Yaskawa INFORM job: A_ROOF_SIDE_0617_2_PAINT_55.JBI

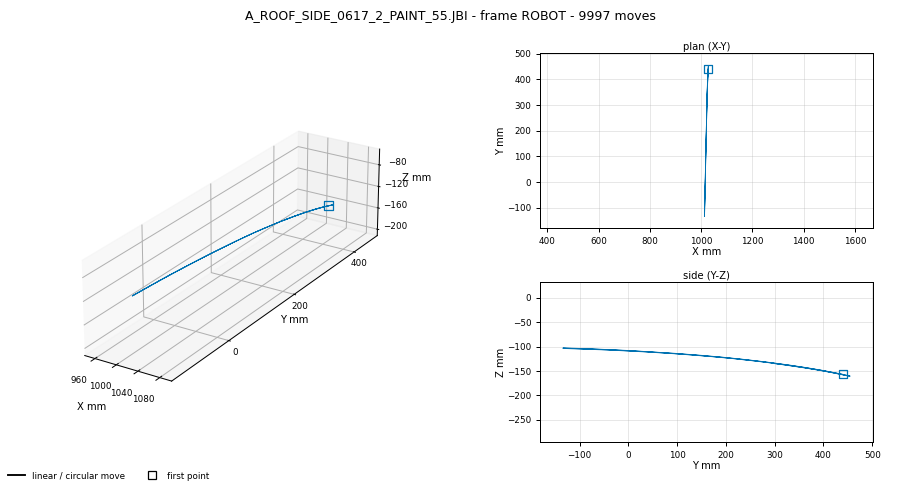
[picture p0: tool path of A_ROOF_SIDE_0617_2_PAINT_55.JBI in frame ROBOT, 9997 of 9997 moves have a stored position in this frame; points joined in program order, loops and branches not executed]
/JOB
//NAME A_ROOF_SIDE_0617_2_PAINT55
//POS
///NPOS 9997,0,0,0,0,0
///TOOL 1
///USER 0
///POSTYPE ROBOT
///RECTAN
///RCONF 1,0,0,0,0,0,0,0,0,0,0,0,0,0,0,0,0,0,0,0,0,0,0,0
C00000=1028.136,439.108,-156.615,175.575,49.117,160.317
C00001=1028.123,438.864,-156.563,175.557,49.112,160.312
C00002=1028.110,438.620,-156.510,175.540,49.107,160.308
C00003=1028.096,438.376,-156.458,175.523,49.102,160.304
C00004=1028.083,438.132,-156.405,175.506,49.097,160.300
C00005=1028.070,437.888,-156.353,175.488,49.092,160.296
C00006=1028.056,437.643,-156.301,175.472,49.087,160.291
C00007=1028.043,437.399,-156.249,175.455,49.082,160.287
C00008=1028.030,437.155,-156.196,175.437,49.078,160.283
C00009=1028.016,436.911,-156.144,175.421,49.072,160.279
C00010=1028.003,436.666,-156.092,175.404,49.067,160.275
C00011=1027.990,436.423,-156.040,175.387,49.063,160.271
C00012=1027.977,436.178,-155.988,175.371,49.057,160.267
C00013=1027.964,435.933,-155.937,175.354,49.053,160.263
C00014=1027.951,435.689,-155.884,175.338,49.048,160.259
C00015=1027.938,435.445,-155.833,175.321,49.043,160.255
C00016=1027.924,435.201,-155.781,175.305,49.038,160.251
C00017=1027.912,434.957,-155.730,175.288,49.034,160.247
C00018=1027.898,434.712,-155.678,175.272,49.029,160.243
C00019=1027.886,434.467,-155.626,175.256,49.025,160.240
C00020=1027.873,434.224,-155.575,175.239,49.020,160.236
C00021=1027.860,433.979,-155.524,175.223,49.015,160.232
C00022=1027.847,433.735,-155.473,175.207,49.010,160.228
C00023=1027.834,433.490,-155.420,175.191,49.006,160.224
C00024=1027.822,433.246,-155.370,175.175,49.001,160.220
C00025=1027.809,433.002,-155.319,175.160,48.997,160.217
C00026=1027.796,432.757,-155.268,175.143,48.992,160.213
C00027=1027.783,432.512,-155.217,175.127,48.988,160.209
C00028=1027.770,432.268,-155.166,175.112,48.983,160.205
C00029=1027.758,432.023,-155.115,175.096,48.979,160.201
C00030=1027.745,431.779,-155.065,175.079,48.974,160.198
C00031=1027.732,431.534,-155.013,175.064,48.969,160.194
C00032=1027.719,431.289,-154.963,175.048,48.965,160.190
C00033=1027.707,431.045,-154.913,175.033,48.961,160.187
C00034=1027.694,430.800,-154.862,175.018,48.956,160.183
C00035=1027.682,430.556,-154.812,175.002,48.952,160.179
C00036=1027.669,430.311,-154.761,174.987,48.947,160.176
C00037=1027.657,430.067,-154.711,174.971,48.943,160.172
C00038=1027.644,429.822,-154.660,174.956,48.939,160.168
C00039=1027.632,429.578,-154.610,174.941,48.934,160.165
C00040=1027.620,429.333,-154.560,174.926,48.930,160.161
C00041=1027.607,429.089,-154.509,174.911,48.926,160.158
C00042=1027.595,428.844,-154.459,174.896,48.921,160.154
C00043=1027.582,428.599,-154.409,174.881,48.917,160.151
C00044=1027.570,428.354,-154.359,174.866,48.913,160.147
C00045=1027.558,428.109,-154.309,174.851,48.908,160.144
C00046=1027.545,427.864,-154.258,174.836,48.904,160.140
C00047=1027.534,427.620,-154.209,174.822,48.900,160.137
C00048=1027.521,427.375,-154.159,174.807,48.896,160.133
C00049=1027.509,427.131,-154.109,174.792,48.892,160.130
C00050=1027.498,426.886,-154.060,174.777,48.888,160.126
C00051=1027.485,426.641,-154.009,174.763,48.884,160.123
C00052=1027.473,426.396,-153.959,174.748,48.880,160.120
C00053=1027.462,426.152,-153.910,174.733,48.876,160.116
C00054=1027.449,425.907,-153.860,174.719,48.872,160.113
C00055=1027.437,425.661,-153.811,174.704,48.868,160.110
C00056=1027.423,425.354,-153.749,174.687,48.862,160.105
C00057=1027.407,425.047,-153.687,174.668,48.858,160.101
C00058=1027.392,424.739,-153.626,174.650,48.853,160.097
C00059=1027.378,424.432,-153.564,174.632,48.847,160.093
C00060=1027.366,424.188,-153.514,174.618,48.843,160.089
C00061=1027.353,423.943,-153.465,174.604,48.840,160.086
C00062=1027.342,423.698,-153.416,174.590,48.835,160.083
C00063=1027.330,423.453,-153.367,174.576,48.832,160.080
C00064=1027.319,423.208,-153.318,174.562,48.828,160.077
C00065=1027.307,422.963,-153.269,174.548,48.824,160.073
C00066=1027.295,422.718,-153.221,174.534,48.820,160.070
C00067=1027.283,422.473,-153.172,174.520,48.817,160.067
C00068=1027.272,422.228,-153.123,174.506,48.813,160.064
C00069=1027.260,421.984,-153.074,174.493,48.809,160.061
C00070=1027.248,421.738,-153.026,174.478,48.806,160.058
C00071=1027.237,421.493,-152.977,174.465,48.802,160.055
C00072=1027.225,421.248,-152.929,174.451,48.798,160.051
C00073=1027.213,421.003,-152.880,174.438,48.794,160.048
C00074=1027.202,420.758,-152.832,174.424,48.790,160.045
C00075=1027.190,420.512,-152.784,174.410,48.787,160.042
C00076=1027.178,420.267,-152.735,174.397,48.783,160.039
C00077=1027.167,420.022,-152.687,174.384,48.779,160.036
C00078=1027.156,419.777,-152.639,174.370,48.776,160.033
C00079=1027.144,419.532,-152.591,174.357,48.773,160.030
C00080=1027.133,419.286,-152.543,174.344,48.769,160.027
C00081=1027.121,419.042,-152.495,174.330,48.766,160.024
C00082=1027.110,418.797,-152.446,174.316,48.762,160.021
C00083=1027.099,418.551,-152.399,174.304,48.758,160.018
C00084=1027.087,418.306,-152.351,174.290,48.754,160.015
C00085=1027.076,418.061,-152.303,174.277,48.751,160.012
C00086=1027.064,417.816,-152.255,174.265,48.748,160.009
C00087=1027.054,417.571,-152.207,174.252,48.744,160.006
C00088=1027.042,417.326,-152.159,174.238,48.741,160.003
C00089=1027.031,417.081,-152.111,174.225,48.737,160.000
C00090=1027.021,416.836,-152.064,174.212,48.734,159.997
C00091=1027.009,416.590,-152.016,174.199,48.730,159.994
C00092=1026.998,416.345,-151.968,174.186,48.727,159.992
C00093=1026.987,416.100,-151.921,174.173,48.724,159.989
C00094=1026.976,415.855,-151.873,174.161,48.721,159.986
C00095=1026.964,415.609,-151.826,174.149,48.717,159.983
C00096=1026.953,415.364,-151.779,174.136,48.714,159.980
C00097=1026.943,415.118,-151.732,174.123,48.710,159.978
C00098=1026.931,414.874,-151.684,174.110,48.707,159.975
C00099=1026.920,414.628,-151.637,174.097,48.704,159.972
C00100=1026.909,414.383,-151.591,174.085,48.701,159.969
C00101=1026.898,414.137,-151.543,174.072,48.698,159.966
C00102=1026.887,413.892,-151.496,174.060,48.695,159.964
C00103=1026.876,413.647,-151.449,174.048,48.691,159.961
C00104=1026.865,413.401,-151.402,174.035,48.688,159.958
C00105=1026.854,413.156,-151.356,174.022,48.685,159.955
C00106=1026.843,412.911,-151.309,174.010,48.682,159.953
C00107=1026.833,412.665,-151.261,173.998,48.679,159.950
C00108=1026.822,412.442,-151.219,173.987,48.676,159.948
C00109=1026.813,412.219,-151.176,173.976,48.673,159.945
C00110=1026.802,411.995,-151.134,173.964,48.670,159.943
C00111=1026.793,411.772,-151.092,173.953,48.668,159.940
C00112=1026.783,411.549,-151.050,173.942,48.665,159.938
C00113=1026.773,411.325,-151.006,173.931,48.662,159.935
C00114=1026.764,411.102,-150.964,173.920,48.659,159.933
C00115=1026.754,410.878,-150.922,173.909,48.656,159.931
C00116=1026.739,410.537,-150.857,173.893,48.653,159.927
C00117=1026.725,410.198,-150.793,173.876,48.648,159.924
C00118=1026.710,409.856,-150.729,173.859,48.644,159.920
C00119=1026.695,409.516,-150.664,173.843,48.640,159.916
C00120=1026.685,409.270,-150.619,173.831,48.637,159.914
C00121=1026.674,409.024,-150.573,173.820,48.634,159.911
C00122=1026.663,408.779,-150.527,173.807,48.632,159.909
C00123=1026.653,408.533,-150.481,173.796,48.629,159.906
C00124=1026.642,408.288,-150.435,173.783,48.626,159.904
C00125=1026.632,408.042,-150.389,173.772,48.623,159.901
C00126=1026.621,407.797,-150.343,173.761,48.620,159.899
C00127=1026.610,407.551,-150.297,173.749,48.618,159.896
C00128=1026.600,407.305,-150.251,173.737,48.615,159.894
C00129=1026.589,407.060,-150.205,173.726,48.612,159.891
C00130=1026.578,406.815,-150.160,173.714,48.609,159.889
C00131=1026.568,406.570,-150.115,173.703,48.607,159.887
C00132=1026.557,406.323,-150.069,173.691,48.604,159.884
C00133=1026.547,406.078,-150.023,173.680,48.601,159.882
C00134=1026.537,405.833,-149.978,173.668,48.599,159.879
C00135=1026.526,405.587,-149.933,173.657,48.596,159.877
C00136=1026.516,405.341,-149.887,173.646,48.594,159.875
C00137=1026.506,405.096,-149.842,173.635,48.591,159.872
C00138=1026.495,404.850,-149.796,173.624,48.588,159.870
C00139=1026.486,404.604,-149.751,173.612,48.585,159.867
C00140=1026.475,404.359,-149.705,173.600,48.583,159.865
C00141=1026.465,404.113,-149.661,173.589,48.580,159.863
C00142=1026.455,403.868,-149.615,173.578,48.578,159.860
C00143=1026.445,403.622,-149.570,173.567,48.576,159.858
C00144=1026.435,403.376,-149.525,173.556,48.573,159.856
C00145=1026.425,403.131,-149.479,173.545,48.570,159.853
C00146=1026.414,402.885,-149.434,173.534,48.568,159.851
C00147=1026.405,402.639,-149.389,173.523,48.565,159.849
C00148=1026.395,402.394,-149.344,173.512,48.562,159.846
C00149=1026.385,402.148,-149.299,173.501,48.560,159.844
C00150=1026.375,401.902,-149.254,173.490,48.558,159.842
C00151=1026.365,401.657,-149.209,173.479,48.555,159.840
C00152=1026.354,401.411,-149.165,173.468,48.553,159.838
C00153=1026.344,401.165,-149.120,173.457,48.551,159.835
C00154=1026.335,400.920,-149.075,173.446,48.548,159.833
C00155=1026.324,400.673,-149.030,173.435,48.546,159.831
C00156=1026.315,400.428,-148.985,173.425,48.543,159.829
C00157=1026.305,400.182,-148.942,173.415,48.541,159.826
C00158=1026.295,399.937,-148.897,173.404,48.539,159.824
C00159=1026.285,399.691,-148.852,173.393,48.537,159.822
C00160=1026.275,399.444,-148.807,173.382,48.535,159.820
C00161=1026.265,399.199,-148.763,173.371,48.532,159.818
C00162=1026.255,398.953,-148.719,173.361,48.530,159.816
C00163=1026.246,398.707,-148.674,173.351,48.528,159.813
C00164=1026.235,398.462,-148.631,173.340,48.525,159.811
C00165=1026.226,398.216,-148.586,173.329,48.523,159.809
C00166=1026.216,397.970,-148.542,173.318,48.521,159.807
C00167=1026.206,397.725,-148.498,173.309,48.519,159.805
C00168=1026.196,397.479,-148.454,173.298,48.517,159.803
C00169=1026.186,397.233,-148.410,173.287,48.515,159.801
C00170=1026.177,396.987,-148.366,173.277,48.513,159.799
C00171=1026.167,396.741,-148.322,173.267,48.510,159.796
C00172=1026.157,396.495,-148.278,173.256,48.509,159.794
C00173=1026.147,396.250,-148.234,173.246,48.506,159.792
C00174=1026.137,396.003,-148.190,173.236,48.504,159.790
C00175=1026.127,395.758,-148.146,173.225,48.502,159.788
C00176=1026.117,395.483,-148.097,173.215,48.500,159.786
C00177=1026.106,395.209,-148.049,173.203,48.498,159.784
C00178=1026.096,394.934,-148.000,173.192,48.495,159.782
C00179=1026.084,394.660,-147.951,173.180,48.493,159.779
C00180=1026.075,394.413,-147.908,173.170,48.491,159.777
C00181=1026.065,394.168,-147.865,173.160,48.489,159.775
C00182=1026.056,393.922,-147.820,173.150,48.487,159.773
C00183=1026.046,393.676,-147.777,173.140,48.485,159.771
C00184=1026.037,393.430,-147.734,173.130,48.483,159.769
C00185=1026.027,393.184,-147.690,173.120,48.482,159.767
C00186=1026.018,392.938,-147.646,173.110,48.480,159.765
C00187=1026.008,392.691,-147.604,173.100,48.478,159.764
C00188=1025.999,392.446,-147.560,173.090,48.476,159.762
C00189=1025.989,392.199,-147.517,173.080,48.474,159.760
C00190=1025.979,391.954,-147.473,173.070,48.472,159.758
C00191=1025.971,391.707,-147.430,173.060,48.471,159.756
C00192=1025.961,391.461,-147.388,173.051,48.469,159.754
C00193=1025.951,391.216,-147.344,173.040,48.467,159.752
C00194=1025.942,390.969,-147.301,173.031,48.465,159.750
C00195=1025.933,390.723,-147.259,173.021,48.463,159.748
C00196=1025.923,390.477,-147.216,173.011,48.462,159.746
C00197=1025.914,390.232,-147.172,173.002,48.460,159.745
C00198=1025.905,389.985,-147.129,172.992,48.458,159.743
C00199=1025.895,389.739,-147.087,172.982,48.457,159.741
C00200=1025.886,389.493,-147.043,172.973,48.455,159.739
C00201=1025.877,389.247,-147.001,172.963,48.453,159.737
C00202=1025.868,389.001,-146.959,172.953,48.452,159.735
C00203=1025.858,388.755,-146.916,172.944,48.450,159.733
C00204=1025.849,388.509,-146.873,172.935,48.448,159.732
C00205=1025.840,388.262,-146.830,172.925,48.446,159.730
C00206=1025.830,388.016,-146.788,172.915,48.445,159.728
C00207=1025.821,387.771,-146.745,172.906,48.443,159.726
C00208=1025.812,387.524,-146.703,172.896,48.442,159.724
C00209=1025.802,387.278,-146.661,172.887,48.440,159.723
C00210=1025.794,387.032,-146.618,172.877,48.439,159.721
C00211=1025.785,386.786,-146.575,172.868,48.437,159.719
C00212=1025.775,386.539,-146.533,172.859,48.436,159.717
C00213=1025.766,386.293,-146.491,172.849,48.434,159.716
C00214=1025.757,386.047,-146.449,172.840,48.433,159.714
C00215=1025.748,385.801,-146.406,172.830,48.431,159.712
C00216=1025.738,385.554,-146.364,172.821,48.430,159.710
C00217=1025.729,385.308,-146.322,172.812,48.429,159.709
C00218=1025.720,385.062,-146.280,172.803,48.427,159.707
C00219=1025.711,384.816,-146.239,172.794,48.426,159.705
C00220=1025.702,384.570,-146.196,172.785,48.424,159.704
C00221=1025.693,384.323,-146.154,172.776,48.423,159.702
C00222=1025.684,384.077,-146.113,172.767,48.422,159.700
C00223=1025.674,383.830,-146.071,172.757,48.421,159.699
C00224=1025.665,383.584,-146.028,172.748,48.419,159.697
C00225=1025.655,383.338,-145.987,172.738,48.418,159.695
C00226=1025.646,383.092,-145.945,172.729,48.416,159.694
C00227=1025.638,382.846,-145.904,172.720,48.415,159.692
C00228=1025.629,382.599,-145.862,172.711,48.413,159.690
C00229=1025.620,382.353,-145.820,172.702,48.413,159.689
C00230=1025.611,382.106,-145.778,172.693,48.411,159.687
C00231=1025.602,381.860,-145.737,172.684,48.410,159.685
C00232=1025.593,381.618,-145.696,172.676,48.409,159.684
C00233=1025.585,381.376,-145.655,172.667,48.408,159.682
C00234=1025.575,381.133,-145.614,172.658,48.406,159.681
C00235=1025.567,380.892,-145.573,172.650,48.405,159.679
C00236=1025.558,380.649,-145.533,172.641,48.404,159.677
C00237=1025.550,380.408,-145.492,172.632,48.403,159.676
C00238=1025.540,380.165,-145.451,172.623,48.401,159.674
C00239=1025.532,379.923,-145.411,172.615,48.400,159.673
C00240=1025.523,379.677,-145.369,172.606,48.399,159.671
C00241=1025.514,379.430,-145.327,172.597,48.398,159.670
C00242=1025.506,379.185,-145.286,172.589,48.397,159.668
C00243=1025.497,378.938,-145.245,172.579,48.396,159.667
C00244=1025.488,378.691,-145.203,172.571,48.395,159.665
C00245=1025.480,378.444,-145.162,172.562,48.394,159.664
C00246=1025.471,378.199,-145.121,172.553,48.393,159.662
C00247=1025.463,377.952,-145.080,172.545,48.391,159.661
C00248=1025.454,377.705,-145.038,172.536,48.391,159.659
C00249=1025.445,377.459,-144.998,172.527,48.389,159.657
C00250=1025.436,377.213,-144.957,172.519,48.388,159.656
C00251=1025.428,376.966,-144.916,172.510,48.387,159.654
C00252=1025.419,376.720,-144.874,172.502,48.386,159.653
C00253=1025.411,376.473,-144.833,172.493,48.385,159.652
C00254=1025.401,376.227,-144.793,172.485,48.385,159.650
C00255=1025.393,375.980,-144.752,172.476,48.384,159.649
C00256=1025.384,375.734,-144.712,172.468,48.383,159.647
C00257=1025.376,375.487,-144.671,172.460,48.382,159.646
C00258=1025.366,375.241,-144.631,172.451,48.381,159.644
C00259=1025.358,374.994,-144.590,172.442,48.380,159.643
C00260=1025.350,374.747,-144.549,172.434,48.379,159.641
C00261=1025.340,374.501,-144.509,172.426,48.378,159.640
C00262=1025.332,374.254,-144.468,172.417,48.377,159.638
C00263=1025.324,374.008,-144.428,172.408,48.376,159.637
C00264=1025.315,373.761,-144.387,172.401,48.376,159.636
C00265=1025.306,373.515,-144.347,172.392,48.375,159.634
C00266=1025.298,373.268,-144.306,172.383,48.374,159.633
C00267=1025.290,373.022,-144.265,172.376,48.373,159.631
C00268=1025.281,372.775,-144.226,172.367,48.373,159.630
C00269=1025.272,372.529,-144.185,172.358,48.372,159.629
C00270=1025.264,372.283,-144.145,172.351,48.371,159.627
C00271=1025.255,372.036,-144.104,172.342,48.370,159.626
C00272=1025.247,371.789,-144.065,172.335,48.369,159.624
C00273=1025.239,371.543,-144.024,172.326,48.369,159.623
C00274=1025.229,371.296,-143.984,172.318,48.368,159.622
C00275=1025.222,371.049,-143.944,172.310,48.367,159.620
C00276=1025.213,370.803,-143.903,172.301,48.367,159.619
C00277=1025.204,370.556,-143.863,172.294,48.366,159.618
C00278=1025.196,370.309,-143.823,172.285,48.365,159.616
C00279=1025.188,370.063,-143.783,172.277,48.365,159.615
C00280=1025.180,369.816,-143.743,172.269,48.364,159.614
C00281=1025.171,369.570,-143.703,172.261,48.363,159.612
C00282=1025.163,369.323,-143.662,172.253,48.362,159.611
C00283=1025.154,369.076,-143.623,172.245,48.362,159.610
C00284=1025.147,368.829,-143.583,172.237,48.361,159.608
C00285=1025.139,368.583,-143.543,172.229,48.361,159.607
C00286=1025.130,368.336,-143.503,172.221,48.360,159.606
C00287=1025.122,368.090,-143.464,172.213,48.360,159.605
C00288=1025.113,367.843,-143.424,172.205,48.359,159.603
C00289=1025.105,367.596,-143.384,172.197,48.359,159.602
C00290=1025.096,367.349,-143.345,172.190,48.358,159.601
C00291=1025.088,367.102,-143.306,172.181,48.358,159.600
C00292=1025.080,366.871,-143.269,172.174,48.357,159.598
C00293=1025.072,366.640,-143.231,172.166,48.357,159.597
C00294=1025.065,366.408,-143.195,172.159,48.356,159.596
C00295=1025.056,366.177,-143.157,172.152,48.356,159.595
C00296=1025.049,365.946,-143.120,172.145,48.356,159.594
C00297=1025.041,365.714,-143.083,172.137,48.355,159.592
C00298=1025.033,365.483,-143.046,172.130,48.355,159.591
C00299=1025.026,365.251,-143.009,172.123,48.354,159.590
C00300=1025.017,365.004,-142.970,172.115,48.354,159.589
C00301=1025.009,364.757,-142.931,172.107,48.353,159.588
C00302=1025.000,364.511,-142.891,172.100,48.353,159.587
C00303=1024.993,364.263,-142.852,172.091,48.353,159.585
C00304=1024.985,364.017,-142.813,172.084,48.353,159.584
C00305=1024.977,363.771,-142.774,172.077,48.352,159.583
C00306=1024.968,363.524,-142.735,172.068,48.352,159.582
C00307=1024.960,363.277,-142.696,172.061,48.351,159.581
C00308=1024.952,363.030,-142.656,172.054,48.351,159.580
C00309=1024.944,362.783,-142.617,172.046,48.351,159.578
C00310=1024.936,362.536,-142.578,172.038,48.350,159.577
C00311=1024.927,362.290,-142.539,172.031,48.350,159.576
C00312=1024.920,362.043,-142.501,172.023,48.350,159.575
C00313=1024.912,361.796,-142.461,172.015,48.349,159.574
C00314=1024.904,361.549,-142.422,172.008,48.349,159.573
C00315=1024.895,361.302,-142.383,172.000,48.349,159.571
C00316=1024.888,361.056,-142.344,171.993,48.349,159.570
C00317=1024.881,360.808,-142.305,171.986,48.348,159.569
C00318=1024.872,360.562,-142.266,171.979,48.349,159.568
C00319=1024.865,360.315,-142.228,171.970,48.348,159.567
C00320=1024.856,360.068,-142.189,171.963,48.348,159.566
C00321=1024.848,359.821,-142.150,171.956,48.348,159.565
C00322=1024.840,359.574,-142.111,171.949,48.348,159.564
C00323=1024.832,359.328,-142.073,171.941,48.348,159.562
C00324=1024.824,359.080,-142.034,171.933,48.347,159.561
C00325=1024.816,358.833,-141.996,171.926,48.347,159.560
C00326=1024.808,358.587,-141.957,171.919,48.347,159.559
C00327=1024.800,358.340,-141.919,171.911,48.348,159.558
C00328=1024.792,358.092,-141.880,171.904,48.347,159.557
C00329=1024.784,357.846,-141.843,171.897,48.347,159.556
C00330=1024.776,357.599,-141.804,171.890,48.347,159.555
C00331=1024.768,357.352,-141.766,171.882,48.347,159.554
C00332=1024.760,357.105,-141.727,171.875,48.347,159.553
C00333=1024.752,356.859,-141.689,171.868,48.347,159.552
C00334=1024.744,356.611,-141.650,171.860,48.347,159.551
C00335=1024.736,356.364,-141.612,171.853,48.347,159.550
C00336=1024.728,356.118,-141.573,171.846,48.347,159.549
C00337=1024.720,355.870,-141.536,171.838,48.347,159.548
C00338=1024.712,355.624,-141.498,171.831,48.347,159.546
C00339=1024.705,355.377,-141.460,171.824,48.347,159.545
C00340=1024.697,355.130,-141.421,171.817,48.348,159.545
C00341=1024.689,354.883,-141.384,171.810,48.348,159.544
C00342=1024.681,354.636,-141.345,171.803,48.348,159.543
C00343=1024.674,354.389,-141.307,171.796,48.348,159.542
C00344=1024.665,354.142,-141.269,171.788,48.348,159.541
C00345=1024.658,353.895,-141.231,171.781,48.348,159.540
C00346=1024.650,353.647,-141.193,171.774,48.348,159.539
C00347=1024.641,353.401,-141.156,171.767,48.348,159.538
C00348=1024.634,353.154,-141.118,171.760,48.348,159.537
C00349=1024.626,352.907,-141.079,171.753,48.348,159.536
C00350=1024.618,352.660,-141.043,171.746,48.348,159.535
C00351=1024.611,352.413,-141.005,171.739,48.349,159.534
C00352=1024.603,352.184,-140.970,171.732,48.349,159.533
C00353=1024.596,351.956,-140.935,171.726,48.350,159.532
C00354=1024.589,351.728,-140.900,171.720,48.349,159.531
C00355=1024.582,351.500,-140.865,171.713,48.350,159.530
C00356=1024.575,351.272,-140.831,171.707,48.350,159.529
C00357=1024.568,351.044,-140.796,171.700,48.350,159.529
C00358=1024.561,350.816,-140.761,171.693,48.351,159.528
C00359=1024.553,350.588,-140.726,171.687,48.350,159.527
C00360=1024.545,350.340,-140.689,171.681,48.351,159.526
C00361=1024.538,350.093,-140.651,171.674,48.351,159.525
C00362=1024.530,349.847,-140.614,171.667,48.352,159.524
C00363=1024.522,349.599,-140.576,171.660,48.352,159.523
C00364=1024.515,349.352,-140.538,171.653,48.352,159.522
C00365=1024.507,349.105,-140.501,171.646,48.352,159.521
C00366=1024.500,348.858,-140.464,171.639,48.353,159.520
C00367=1024.492,348.611,-140.426,171.632,48.353,159.519
C00368=1024.484,348.364,-140.389,171.626,48.353,159.519
C00369=1024.477,348.117,-140.352,171.619,48.354,159.518
C00370=1024.469,347.870,-140.315,171.612,48.354,159.517
C00371=1024.461,347.622,-140.277,171.605,48.355,159.516
C00372=1024.453,347.376,-140.240,171.599,48.355,159.515
C00373=1024.446,347.128,-140.203,171.591,48.355,159.514
C00374=1024.438,346.881,-140.166,171.585,48.356,159.513
C00375=1024.431,346.634,-140.129,171.578,48.356,159.512
C00376=1024.423,346.387,-140.092,171.571,48.357,159.512
C00377=1024.415,346.140,-140.055,171.565,48.358,159.511
C00378=1024.408,345.893,-140.018,171.558,48.358,159.510
C00379=1024.400,345.646,-139.981,171.551,48.358,159.509
C00380=1024.393,345.399,-139.944,171.544,48.359,159.508
C00381=1024.385,345.151,-139.907,171.537,48.359,159.507
C00382=1024.377,344.904,-139.871,171.531,48.360,159.507
C00383=1024.370,344.657,-139.833,171.524,48.361,159.506
C00384=1024.362,344.410,-139.797,171.518,48.361,159.505
C00385=1024.355,344.163,-139.759,171.512,48.361,159.504
C00386=1024.348,343.915,-139.723,171.505,48.362,159.503
C00387=1024.340,343.668,-139.686,171.498,48.363,159.503
C00388=1024.333,343.421,-139.649,171.492,48.363,159.502
C00389=1024.325,343.174,-139.612,171.485,48.364,159.501
C00390=1024.317,342.926,-139.576,171.478,48.364,159.500
C00391=1024.310,342.680,-139.539,171.471,48.365,159.499
C00392=1024.303,342.432,-139.503,171.465,48.366,159.498
C00393=1024.295,342.185,-139.467,171.459,48.366,159.498
C00394=1024.288,341.938,-139.429,171.453,48.367,159.497
C00395=1024.280,341.690,-139.393,171.446,48.368,159.496
C00396=1024.272,341.443,-139.357,171.439,48.368,159.495
C00397=1024.266,341.196,-139.319,171.432,48.369,159.495
C00398=1024.258,340.949,-139.283,171.426,48.369,159.494
C00399=1024.250,340.702,-139.247,171.419,48.371,159.493
C00400=1024.243,340.454,-139.211,171.414,48.371,159.492
C00401=1024.235,340.207,-139.173,171.407,48.372,159.492
C00402=1024.228,339.960,-139.137,171.400,48.372,159.491
C00403=1024.221,339.713,-139.101,171.394,48.373,159.490
C00404=1024.213,339.465,-139.065,171.387,48.374,159.489
C00405=1024.205,339.218,-139.029,171.380,48.374,159.488
C00406=1024.198,338.971,-138.993,171.375,48.375,159.488
C00407=1024.191,338.723,-138.956,171.368,48.376,159.487
C00408=1024.184,338.476,-138.920,171.362,48.377,159.486
C00409=1024.177,338.229,-138.884,171.355,48.378,159.486
C00410=1024.169,337.982,-138.848,171.349,48.379,159.485
C00411=1024.161,337.734,-138.812,171.343,48.379,159.484
C00412=1024.154,337.505,-138.778,171.337,48.380,159.484
C00413=1024.147,337.275,-138.745,171.331,48.381,159.483
C00414=1024.141,337.045,-138.712,171.325,48.382,159.482
C00415=1024.134,336.816,-138.679,171.319,48.383,159.482
C00416=1024.127,336.586,-138.645,171.314,48.383,159.481
C00417=1024.120,336.356,-138.611,171.307,48.384,159.480
C00418=1024.113,336.126,-138.578,171.302,48.385,159.480
C00419=1024.107,335.897,-138.544,171.297,48.386,159.479
C00420=1024.100,335.649,-138.509,171.290,48.387,159.478
C00421=1024.092,335.402,-138.473,171.284,48.388,159.478
C00422=1024.085,335.155,-138.437,171.277,48.389,159.477
C00423=1024.077,334.907,-138.401,171.271,48.389,159.476
C00424=1024.071,334.660,-138.365,171.265,48.391,159.476
C00425=1024.063,334.413,-138.329,171.259,48.392,159.475
C00426=1024.056,334.165,-138.294,171.252,48.392,159.474
C00427=1024.048,333.918,-138.258,171.247,48.393,159.474
C00428=1024.041,333.671,-138.222,171.240,48.395,159.473
C00429=1024.034,333.423,-138.187,171.234,48.396,159.472
C00430=1024.027,333.176,-138.151,171.228,48.397,159.472
C00431=1024.020,332.928,-138.115,171.222,48.397,159.471
C00432=1024.012,332.682,-138.080,171.215,48.398,159.470
C00433=1024.005,332.434,-138.045,171.209,48.400,159.470
C00434=1023.998,332.186,-138.009,171.204,48.401,159.469
C00435=1023.991,331.940,-137.973,171.197,48.402,159.469
C00436=1023.983,331.692,-137.938,171.191,48.403,159.468
C00437=1023.976,331.445,-137.903,171.185,48.404,159.467
C00438=1023.968,331.197,-137.867,171.179,48.405,159.467
C00439=1023.961,330.950,-137.832,171.173,48.406,159.466
C00440=1023.954,330.702,-137.797,171.166,48.408,159.466
C00441=1023.947,330.454,-137.761,171.161,48.408,159.465
C00442=1023.939,330.208,-137.726,171.155,48.410,159.464
C00443=1023.932,329.960,-137.691,171.148,48.411,159.464
C00444=1023.925,329.712,-137.656,171.143,48.412,159.463
C00445=1023.918,329.465,-137.620,171.137,48.413,159.463
C00446=1023.911,329.218,-137.586,171.131,48.415,159.462
C00447=1023.903,328.970,-137.550,171.125,48.416,159.462
C00448=1023.896,328.723,-137.514,171.119,48.417,159.461
C00449=1023.890,328.476,-137.479,171.112,48.418,159.460
C00450=1023.883,328.228,-137.444,171.107,48.419,159.460
C00451=1023.875,327.981,-137.409,171.101,48.420,159.459
C00452=1023.868,327.733,-137.374,171.094,48.421,159.458
C00453=1023.861,327.486,-137.339,171.089,48.423,159.458
C00454=1023.854,327.239,-137.304,171.083,48.424,159.457
C00455=1023.847,326.992,-137.269,171.077,48.425,159.457
C00456=1023.840,326.743,-137.234,171.072,48.427,159.456
C00457=1023.832,326.496,-137.200,171.065,48.428,159.456
C00458=1023.825,326.249,-137.166,171.059,48.429,159.455
C00459=1023.818,326.001,-137.130,171.054,48.431,159.455
C00460=1023.810,325.753,-137.096,171.047,48.432,159.454
C00461=1023.803,325.506,-137.062,171.041,48.434,159.454
C00462=1023.796,325.259,-137.027,171.036,48.435,159.453
C00463=1023.788,325.012,-136.992,171.030,48.437,159.453
C00464=1023.781,324.764,-136.958,171.024,48.438,159.452
C00465=1023.774,324.516,-136.923,171.019,48.439,159.452
C00466=1023.767,324.268,-136.889,171.012,48.441,159.451
C00467=1023.759,324.021,-136.854,171.006,48.442,159.451
C00468=1023.752,323.774,-136.819,171.001,48.444,159.450
C00469=1023.745,323.526,-136.785,170.995,48.445,159.450
C00470=1023.738,323.279,-136.751,170.990,48.447,159.449
C00471=1023.731,323.031,-136.716,170.983,48.448,159.449
C00472=1023.724,322.799,-136.684,170.978,48.449,159.448
C00473=1023.718,322.567,-136.652,170.972,48.451,159.448
C00474=1023.711,322.335,-136.620,170.967,48.452,159.447
C00475=1023.704,322.103,-136.588,170.962,48.454,159.447
C00476=1023.697,321.871,-136.555,170.957,48.455,159.447
C00477=1023.690,321.640,-136.523,170.950,48.456,159.446
C00478=1023.685,321.408,-136.491,170.945,48.458,159.446
C00479=1023.677,321.176,-136.459,170.940,48.459,159.445
C00480=1023.670,320.928,-136.425,170.934,48.461,159.445
C00481=1023.664,320.680,-136.391,170.929,48.462,159.444
C00482=1023.656,320.433,-136.356,170.923,48.464,159.444
C00483=1023.649,320.186,-136.322,170.918,48.465,159.443
C00484=1023.642,319.938,-136.288,170.912,48.467,159.443
C00485=1023.635,319.691,-136.253,170.906,48.468,159.442
C00486=1023.628,319.443,-136.219,170.900,48.470,159.442
C00487=1023.621,319.195,-136.185,170.894,48.472,159.441
C00488=1023.614,318.947,-136.151,170.889,48.473,159.441
C00489=1023.607,318.700,-136.117,170.883,48.475,159.441
C00490=1023.601,318.453,-136.083,170.878,48.477,159.440
C00491=1023.594,318.205,-136.049,170.872,48.479,159.440
C00492=1023.586,317.958,-136.015,170.867,48.480,159.439
C00493=1023.580,317.710,-135.980,170.861,48.481,159.439
C00494=1023.573,317.462,-135.947,170.856,48.483,159.438
C00495=1023.565,317.215,-135.912,170.850,48.485,159.438
C00496=1023.559,316.968,-135.879,170.845,48.486,159.438
C00497=1023.552,316.720,-135.844,170.839,48.488,159.437
C00498=1023.545,316.472,-135.810,170.834,48.490,159.437
C00499=1023.538,316.225,-135.777,170.828,48.491,159.436
C00500=1023.531,315.977,-135.742,170.823,48.493,159.436
C00501=1023.525,315.730,-135.709,170.817,48.495,159.436
C00502=1023.517,315.482,-135.675,170.812,48.496,159.435
C00503=1023.510,315.234,-135.641,170.805,48.498,159.435
C00504=1023.504,314.987,-135.607,170.800,48.500,159.434
C00505=1023.497,314.739,-135.573,170.794,48.502,159.434
C00506=1023.490,314.492,-135.539,170.789,48.503,159.434
C00507=1023.484,314.244,-135.505,170.783,48.505,159.433
C00508=1023.477,313.997,-135.471,170.779,48.507,159.433
C00509=1023.470,313.749,-135.438,170.773,48.509,159.432
C00510=1023.463,313.502,-135.405,170.768,48.510,159.432
C00511=1023.457,313.254,-135.370,170.762,48.512,159.432
C00512=1023.450,313.006,-135.337,170.756,48.514,159.431
C00513=1023.443,312.759,-135.303,170.751,48.515,159.431
C00514=1023.437,312.511,-135.269,170.745,48.517,159.430
C00515=1023.430,312.264,-135.235,170.741,48.519,159.430
C00516=1023.423,312.016,-135.202,170.735,48.521,159.430
C00517=1023.416,311.768,-135.168,170.730,48.523,159.429
C00518=1023.410,311.521,-135.134,170.724,48.525,159.429
C00519=1023.403,311.273,-135.100,170.719,48.527,159.429
C00520=1023.397,311.025,-135.068,170.714,48.528,159.428
C00521=1023.389,310.778,-135.034,170.708,48.530,159.428
C00522=1023.384,310.530,-135.000,170.703,48.532,159.428
C00523=1023.377,310.282,-134.967,170.697,48.534,159.427
C00524=1023.369,310.036,-134.934,170.692,48.536,159.427
C00525=1023.362,309.787,-134.901,170.686,48.538,159.427
C00526=1023.356,309.539,-134.868,170.681,48.540,159.426
C00527=1023.348,309.292,-134.835,170.676,48.542,159.426
C00528=1023.341,309.044,-134.802,170.671,48.544,159.426
C00529=1023.335,308.796,-134.769,170.665,48.546,159.425
C00530=1023.327,308.549,-134.736,170.660,48.548,159.425
C00531=1023.321,308.301,-134.703,170.654,48.550,159.425
C00532=1023.314,308.072,-134.672,170.649,48.552,159.425
C00533=1023.308,307.842,-134.641,170.644,48.554,159.424
C00534=1023.301,307.614,-134.611,170.640,48.556,159.424
C00535=1023.295,307.384,-134.582,170.635,48.558,159.424
C00536=1023.288,307.154,-134.551,170.630,48.560,159.423
C00537=1023.282,306.925,-134.520,170.625,48.562,159.423
C00538=1023.275,306.696,-134.490,170.620,48.563,159.423
C00539=1023.269,306.467,-134.459,170.616,48.566,159.423
C00540=1023.262,306.219,-134.426,170.610,48.568,159.422
C00541=1023.255,305.971,-134.394,170.605,48.570,159.422
C00542=1023.248,305.723,-134.361,170.599,48.572,159.422
C00543=1023.242,305.475,-134.328,170.594,48.574,159.422
C00544=1023.235,305.228,-134.296,170.589,48.577,159.421
C00545=1023.228,304.980,-134.263,170.584,48.579,159.421
C00546=1023.222,304.732,-134.230,170.579,48.580,159.421
C00547=1023.214,304.484,-134.198,170.573,48.583,159.421
C00548=1023.208,304.237,-134.165,170.569,48.585,159.420
C00549=1023.202,303.989,-134.132,170.563,48.588,159.420
C00550=1023.194,303.741,-134.100,170.558,48.590,159.420
C00551=1023.188,303.493,-134.067,170.552,48.592,159.419
C00552=1023.181,303.246,-134.035,170.548,48.594,159.419
C00553=1023.174,302.998,-134.002,170.543,48.596,159.419
C00554=1023.168,302.750,-133.969,170.537,48.598,159.419
C00555=1023.160,302.503,-133.937,170.532,48.601,159.419
C00556=1023.154,302.255,-133.904,170.527,48.603,159.418
C00557=1023.147,302.007,-133.871,170.522,48.605,159.418
C00558=1023.140,301.760,-133.839,170.517,48.607,159.418
C00559=1023.134,301.512,-133.806,170.512,48.610,159.418
C00560=1023.126,301.264,-133.774,170.507,48.612,159.418
C00561=1023.120,301.016,-133.742,170.501,48.615,159.417
C00562=1023.114,300.768,-133.709,170.497,48.617,159.417
C00563=1023.107,300.521,-133.677,170.492,48.619,159.417
C00564=1023.100,300.273,-133.644,170.486,48.621,159.417
C00565=1023.094,300.025,-133.611,170.481,48.624,159.416
C00566=1023.087,299.777,-133.579,170.476,48.626,159.416
C00567=1023.081,299.530,-133.547,170.471,48.628,159.416
C00568=1023.074,299.283,-133.515,170.466,48.630,159.416
C00569=1023.067,299.034,-133.481,170.461,48.633,159.416
C00570=1023.061,298.786,-133.449,170.456,48.635,159.415
C00571=1023.054,298.539,-133.417,170.451,48.637,159.415
C00572=1023.048,298.291,-133.384,170.446,48.640,159.415
C00573=1023.041,298.043,-133.353,170.441,48.642,159.415
C00574=1023.035,297.796,-133.320,170.436,48.644,159.415
C00575=1023.029,297.547,-133.288,170.430,48.647,159.414
C00576=1023.022,297.300,-133.256,170.426,48.649,159.414
C00577=1023.015,297.052,-133.223,170.421,48.652,159.414
C00578=1023.008,296.804,-133.192,170.416,48.654,159.414
C00579=1023.002,296.556,-133.159,170.411,48.656,159.414
C00580=1022.996,296.308,-133.127,170.406,48.658,159.413
C00581=1022.989,296.061,-133.095,170.401,48.661,159.413
C00582=1022.983,295.813,-133.063,170.396,48.663,159.413
C00583=1022.976,295.565,-133.031,170.392,48.666,159.413
C00584=1022.970,295.317,-132.998,170.386,48.668,159.413
C00585=1022.963,295.070,-132.966,170.381,48.670,159.412
C00586=1022.957,294.822,-132.934,170.376,48.673,159.412
C00587=1022.950,294.574,-132.902,170.371,48.676,159.412
C00588=1022.944,294.326,-132.870,170.366,48.678,159.412
C00589=1022.938,294.078,-132.838,170.362,48.680,159.412
C00590=1022.931,293.830,-132.805,170.356,48.683,159.412
C00591=1022.925,293.582,-132.774,170.352,48.685,159.412
C00592=1022.918,293.362,-132.745,170.347,48.688,159.411
C00593=1022.913,293.141,-132.718,170.343,48.690,159.411
C00594=1022.907,292.920,-132.689,170.339,48.692,159.411
C00595=1022.901,292.699,-132.661,170.334,48.695,159.411
C00596=1022.895,292.479,-132.632,170.330,48.697,159.411
C00597=1022.889,292.258,-132.604,170.326,48.699,159.411
C00598=1022.884,292.038,-132.576,170.322,48.701,159.411
C00599=1022.878,291.818,-132.548,170.317,48.704,159.411
C00600=1022.871,291.570,-132.516,170.312,48.706,159.411
C00601=1022.865,291.322,-132.484,170.307,48.709,159.410
C00602=1022.858,291.074,-132.453,170.302,48.712,159.410
C00603=1022.851,290.826,-132.421,170.298,48.715,159.410
C00604=1022.845,290.578,-132.390,170.292,48.717,159.410
C00605=1022.838,290.330,-132.359,170.288,48.720,159.410
C00606=1022.831,290.082,-132.327,170.283,48.722,159.410
C00607=1022.825,289.834,-132.296,170.278,48.725,159.410
C00608=1022.818,289.586,-132.264,170.274,48.728,159.410
C00609=1022.812,289.338,-132.232,170.269,48.730,159.410
C00610=1022.805,289.090,-132.201,170.264,48.733,159.409
C00611=1022.799,288.843,-132.170,170.259,48.736,159.409
C00612=1022.793,288.595,-132.139,170.255,48.738,159.409
C00613=1022.786,288.347,-132.108,170.249,48.742,159.409
C00614=1022.779,288.099,-132.076,170.245,48.744,159.409
C00615=1022.772,287.851,-132.045,170.240,48.747,159.409
C00616=1022.766,287.603,-132.013,170.235,48.750,159.409
C00617=1022.759,287.355,-131.982,170.230,48.753,159.409
C00618=1022.753,287.107,-131.952,170.226,48.755,159.409
C00619=1022.746,286.859,-131.920,170.221,48.758,159.409
C00620=1022.740,286.611,-131.888,170.216,48.761,159.409
C00621=1022.734,286.363,-131.857,170.212,48.764,159.409
C00622=1022.727,286.115,-131.826,170.206,48.767,159.408
C00623=1022.721,285.868,-131.795,170.202,48.769,159.408
C00624=1022.714,285.620,-131.763,170.198,48.772,159.408
C00625=1022.708,285.372,-131.732,170.192,48.775,159.408
C00626=1022.701,285.123,-131.701,170.188,48.778,159.408
C00627=1022.694,284.876,-131.671,170.183,48.780,159.408
C00628=1022.688,284.628,-131.640,170.178,48.784,159.408
C00629=1022.681,284.380,-131.609,170.173,48.786,159.408
C00630=1022.675,284.131,-131.578,170.169,48.789,159.408
C00631=1022.668,283.883,-131.546,170.164,48.792,159.408
C00632=1022.662,283.636,-131.516,170.159,48.795,159.408
C00633=1022.655,283.388,-131.485,170.155,48.798,159.408
C00634=1022.648,283.139,-131.455,170.150,48.802,159.408
C00635=1022.642,282.892,-131.423,170.146,48.805,159.408
C00636=1022.636,282.644,-131.393,170.141,48.808,159.408
C00637=1022.629,282.396,-131.361,170.136,48.811,159.408
C00638=1022.622,282.148,-131.331,170.132,48.814,159.408
C00639=1022.616,281.900,-131.300,170.127,48.816,159.408
C00640=1022.610,281.652,-131.269,170.122,48.820,159.408
C00641=1022.603,281.403,-131.239,170.118,48.822,159.408
C00642=1022.597,281.156,-131.208,170.113,48.825,159.408
C00643=1022.590,280.908,-131.178,170.108,48.828,159.408
C00644=1022.583,280.659,-131.147,170.104,48.831,159.408
C00645=1022.577,280.412,-131.116,170.100,48.835,159.408
C00646=1022.571,280.164,-131.085,170.094,48.838,159.408
C00647=1022.564,279.915,-131.054,170.090,48.841,159.408
C00648=1022.558,279.668,-131.024,170.085,48.844,159.408
C00649=1022.551,279.420,-130.993,170.081,48.846,159.408
C00650=1022.545,279.172,-130.963,170.076,48.850,159.408
C00651=1022.539,278.923,-130.932,170.072,48.853,159.408
C00652=1022.533,278.709,-130.906,170.067,48.856,159.408
C00653=1022.528,278.494,-130.879,170.064,48.858,159.408
C00654=1022.522,278.280,-130.853,170.059,48.861,159.408
C00655=1022.517,278.065,-130.826,170.056,48.863,159.408
C00656=1022.511,277.850,-130.800,170.052,48.866,159.408
C00657=1022.506,277.637,-130.774,170.048,48.869,159.408
C00658=1022.500,277.422,-130.747,170.044,48.871,159.408
C00659=1022.494,277.207,-130.720,170.040,48.874,159.408
C00660=1022.489,276.959,-130.690,170.035,48.877,159.408
C00661=1022.481,276.712,-130.659,170.031,48.881,159.408
C00662=1022.475,276.464,-130.629,170.026,48.884,159.408
C00663=1022.469,276.215,-130.598,170.022,48.887,159.408
C00664=1022.462,275.968,-130.568,170.018,48.890,159.408
C00665=1022.456,275.719,-130.538,170.014,48.894,159.408
C00666=1022.449,275.472,-130.508,170.008,48.897,159.408
C00667=1022.443,275.222,-130.478,170.004,48.900,159.408
C00668=1022.437,274.975,-130.448,170.000,48.903,159.408
C00669=1022.430,274.726,-130.417,169.995,48.906,159.408
C00670=1022.424,274.479,-130.388,169.991,48.910,159.408
C00671=1022.417,274.230,-130.357,169.986,48.913,159.408
C00672=1022.411,273.983,-130.327,169.981,48.916,159.409
C00673=1022.404,273.734,-130.297,169.977,48.919,159.409
C00674=1022.399,273.487,-130.266,169.973,48.923,159.409
C00675=1022.391,273.238,-130.236,169.967,48.926,159.409
C00676=1022.386,272.990,-130.206,169.963,48.929,159.409
C00677=1022.379,272.742,-130.176,169.959,48.932,159.409
C00678=1022.373,272.494,-130.146,169.955,48.936,159.409
C00679=1022.366,272.246,-130.116,169.950,48.940,159.409
C00680=1022.360,271.998,-130.085,169.946,48.942,159.409
C00681=1022.354,271.750,-130.056,169.942,48.946,159.409
C00682=1022.347,271.502,-130.026,169.936,48.949,159.409
C00683=1022.341,271.254,-129.996,169.932,48.953,159.409
C00684=1022.334,271.006,-129.966,169.928,48.956,159.410
C00685=1022.328,270.757,-129.936,169.923,48.959,159.409
C00686=1022.321,270.510,-129.906,169.919,48.963,159.410
C00687=1022.315,270.261,-129.876,169.915,48.966,159.410
C00688=1022.309,270.013,-129.847,169.911,48.969,159.410
C00689=1022.303,269.765,-129.816,169.906,48.973,159.410
C00690=1022.296,269.516,-129.787,169.902,48.977,159.410
C00691=1022.290,269.269,-129.757,169.898,48.980,159.410
C00692=1022.284,269.021,-129.727,169.892,48.983,159.410
C00693=1022.277,268.772,-129.697,169.888,48.987,159.410
C00694=1022.270,268.525,-129.668,169.884,48.990,159.410
C00695=1022.264,268.276,-129.639,169.879,48.994,159.411
C00696=1022.258,268.028,-129.608,169.875,48.998,159.411
C00697=1022.251,267.780,-129.579,169.871,49.001,159.411
C00698=1022.245,267.532,-129.549,169.867,49.004,159.411
C00699=1022.239,267.283,-129.519,169.862,49.008,159.411
C00700=1022.233,267.035,-129.490,169.858,49.011,159.411
C00701=1022.226,266.787,-129.460,169.854,49.015,159.411
C00702=1022.219,266.539,-129.431,169.849,49.019,159.411
C00703=1022.213,266.291,-129.401,169.845,49.022,159.412
C00704=1022.207,266.043,-129.372,169.841,49.026,159.412
C00705=1022.201,265.795,-129.342,169.836,49.029,159.412
C00706=1022.194,265.546,-129.312,169.832,49.033,159.412
C00707=1022.188,265.298,-129.283,169.828,49.037,159.412
C00708=1022.182,265.050,-129.254,169.823,49.040,159.412
C00709=1022.175,264.802,-129.224,169.819,49.044,159.413
C00710=1022.168,264.553,-129.195,169.815,49.047,159.413
C00711=1022.162,264.305,-129.165,169.811,49.051,159.413
C00712=1022.157,264.093,-129.141,169.807,49.054,159.413
C00713=1022.151,263.881,-129.115,169.803,49.057,159.413
C00714=1022.147,263.669,-129.090,169.799,49.060,159.413
C00715=1022.141,263.456,-129.065,169.795,49.063,159.413
C00716=1022.136,263.244,-129.040,169.792,49.067,159.414
C00717=1022.130,263.032,-129.014,169.788,49.069,159.413
C00718=1022.124,262.819,-128.990,169.785,49.073,159.414
C00719=1022.119,262.607,-128.965,169.781,49.076,159.414
C00720=1022.113,262.359,-128.935,169.777,49.080,159.414
C00721=1022.107,262.111,-128.906,169.773,49.083,159.414
C00722=1022.100,261.862,-128.877,169.768,49.087,159.414
C00723=1022.094,261.614,-128.848,169.764,49.091,159.415
C00724=1022.087,261.366,-128.819,169.760,49.094,159.415
C00725=1022.081,261.118,-128.789,169.755,49.098,159.415
C00726=1022.075,260.870,-128.760,169.751,49.101,159.415
C00727=1022.069,260.622,-128.731,169.748,49.106,159.415
C00728=1022.062,260.374,-128.702,169.744,49.109,159.416
C00729=1022.056,260.126,-128.673,169.739,49.113,159.416
C00730=1022.049,259.877,-128.644,169.735,49.117,159.416
C00731=1022.043,259.629,-128.615,169.730,49.121,159.416
C00732=1022.036,259.381,-128.586,169.726,49.125,159.416
C00733=1022.030,259.133,-128.557,169.722,49.129,159.417
C00734=1022.023,258.884,-128.528,169.717,49.133,159.417
C00735=1022.017,258.636,-128.501,169.713,49.136,159.417
C00736=1022.011,258.388,-128.472,169.710,49.140,159.417
C00737=1022.004,258.139,-128.442,169.705,49.144,159.417
C00738=1021.997,257.891,-128.414,169.701,49.148,159.418
C00739=1021.991,257.642,-128.385,169.696,49.152,159.418
C00740=1021.985,257.394,-128.356,169.692,49.156,159.418
C00741=1021.978,257.146,-128.327,169.688,49.160,159.418
C00742=1021.971,256.898,-128.299,169.683,49.164,159.418
C00743=1021.965,256.650,-128.271,169.680,49.168,159.419
C00744=1021.959,256.402,-128.242,169.676,49.172,159.419
C00745=1021.952,256.154,-128.213,169.671,49.176,159.419
C00746=1021.946,255.905,-128.185,169.667,49.180,159.419
C00747=1021.940,255.657,-128.156,169.664,49.184,159.420
C00748=1021.933,255.409,-128.127,169.659,49.188,159.420
C00749=1021.927,255.160,-128.099,169.655,49.192,159.420
C00750=1021.921,254.912,-128.070,169.650,49.196,159.420
C00751=1021.914,254.664,-128.041,169.646,49.200,159.421
C00752=1021.908,254.416,-128.013,169.643,49.204,159.421
C00753=1021.902,254.167,-127.984,169.638,49.208,159.421
C00754=1021.896,253.919,-127.956,169.634,49.212,159.421
C00755=1021.889,253.671,-127.927,169.630,49.216,159.422
C00756=1021.882,253.423,-127.898,169.625,49.220,159.422
C00757=1021.876,253.174,-127.870,169.622,49.224,159.422
C00758=1021.869,252.926,-127.842,169.618,49.228,159.422
C00759=1021.863,252.677,-127.813,169.613,49.232,159.423
C00760=1021.857,252.429,-127.784,169.609,49.236,159.423
C00761=1021.851,252.181,-127.756,169.606,49.240,159.423
C00762=1021.844,251.933,-127.727,169.601,49.245,159.423
C00763=1021.838,251.684,-127.699,169.597,49.248,159.424
C00764=1021.831,251.436,-127.671,169.593,49.252,159.424
C00765=1021.825,251.187,-127.642,169.589,49.257,159.424
C00766=1021.820,250.939,-127.614,169.585,49.260,159.424
C00767=1021.813,250.690,-127.585,169.581,49.265,159.425
C00768=1021.807,250.442,-127.557,169.576,49.269,159.425
C00769=1021.800,250.194,-127.528,169.572,49.273,159.425
C00770=1021.795,249.946,-127.500,169.569,49.277,159.426
C00771=1021.788,249.698,-127.472,169.564,49.281,159.426
C00772=1021.783,249.485,-127.447,169.561,49.285,159.426
C00773=1021.778,249.271,-127.423,169.557,49.288,159.426
C00774=1021.772,249.058,-127.398,169.555,49.292,159.427
C00775=1021.767,248.846,-127.375,169.551,49.296,159.427
C00776=1021.761,248.632,-127.351,169.547,49.299,159.427
C00777=1021.756,248.419,-127.326,169.544,49.302,159.427
C00778=1021.751,248.206,-127.301,169.540,49.306,159.428
C00779=1021.746,247.993,-127.277,169.537,49.310,159.428
C00780=1021.739,247.745,-127.249,169.532,49.314,159.428
C00781=1021.733,247.496,-127.221,169.528,49.318,159.428
C00782=1021.727,247.248,-127.192,169.525,49.322,159.429
C00783=1021.721,246.999,-127.165,169.520,49.327,159.429
C00784=1021.715,246.752,-127.136,169.517,49.331,159.429
C00785=1021.709,246.503,-127.108,169.513,49.335,159.430
C00786=1021.702,246.255,-127.080,169.508,49.339,159.430
C00787=1021.696,246.006,-127.051,169.504,49.343,159.430
C00788=1021.691,245.758,-127.023,169.501,49.348,159.431
C00789=1021.684,245.510,-126.995,169.496,49.352,159.431
C00790=1021.678,245.261,-126.967,169.492,49.356,159.431
C00791=1021.672,245.012,-126.938,169.489,49.360,159.432
C00792=1021.666,244.765,-126.911,169.485,49.365,159.432
C00793=1021.660,244.517,-126.882,169.481,49.369,159.432
C00794=1021.654,244.268,-126.854,169.477,49.373,159.432
C00795=1021.647,244.019,-126.826,169.473,49.377,159.433
C00796=1021.642,243.771,-126.798,169.468,49.382,159.433
C00797=1021.636,243.523,-126.770,169.465,49.386,159.433
C00798=1021.629,243.274,-126.742,169.461,49.390,159.434
C00799=1021.623,243.026,-126.715,169.457,49.395,159.434
C00800=1021.617,242.778,-126.686,169.453,49.399,159.434
C00801=1021.610,242.529,-126.659,169.449,49.404,159.435
C00802=1021.604,242.281,-126.631,169.445,49.408,159.435
C00803=1021.598,242.033,-126.603,169.441,49.412,159.435
C00804=1021.592,241.784,-126.575,169.437,49.417,159.436
C00805=1021.586,241.535,-126.547,169.433,49.421,159.436
C00806=1021.580,241.288,-126.519,169.430,49.425,159.436
C00807=1021.573,241.039,-126.492,169.425,49.430,159.437
C00808=1021.567,240.791,-126.463,169.421,49.434,159.437
C00809=1021.561,240.543,-126.436,169.418,49.439,159.438
C00810=1021.555,240.293,-126.408,169.413,49.444,159.438
C00811=1021.549,240.045,-126.381,169.410,49.448,159.438
C00812=1021.543,239.797,-126.353,169.405,49.452,159.439
C00813=1021.537,239.548,-126.325,169.402,49.457,159.439
C00814=1021.530,239.300,-126.297,169.398,49.462,159.439
C00815=1021.524,239.052,-126.271,169.394,49.466,159.440
C00816=1021.518,238.803,-126.243,169.390,49.470,159.440
C00817=1021.511,238.556,-126.216,169.385,49.475,159.440
C00818=1021.505,238.307,-126.188,169.382,49.480,159.441
C00819=1021.499,238.058,-126.160,169.379,49.484,159.441
C00820=1021.493,237.810,-126.133,169.374,49.489,159.442
C00821=1021.486,237.562,-126.105,169.371,49.493,159.442
C00822=1021.480,237.312,-126.078,169.366,49.498,159.442
C00823=1021.474,237.065,-126.051,169.363,49.503,159.443
C00824=1021.468,236.816,-126.024,169.359,49.507,159.443
C00825=1021.461,236.568,-125.996,169.355,49.512,159.443
C00826=1021.455,236.319,-125.969,169.351,49.517,159.444
C00827=1021.448,236.070,-125.942,169.347,49.521,159.444
C00828=1021.442,235.823,-125.914,169.344,49.526,159.445
C00829=1021.436,235.574,-125.887,169.339,49.531,159.445
C00830=1021.431,235.326,-125.859,169.336,49.536,159.446
C00831=1021.424,235.076,-125.832,169.332,49.540,159.446
C00832=1021.418,234.860,-125.809,169.328,49.544,159.446
C00833=1021.413,234.644,-125.785,169.325,49.548,159.447
C00834=1021.408,234.428,-125.761,169.321,49.553,159.447
C00835=1021.402,234.212,-125.738,169.319,49.556,159.448
C00836=1021.397,233.996,-125.714,169.315,49.561,159.448
C00837=1021.392,233.779,-125.690,169.311,49.565,159.448
C00838=1021.386,233.563,-125.666,169.308,49.569,159.449
C00839=1021.380,233.347,-125.643,169.305,49.573,159.449
C00840=1021.375,233.098,-125.616,169.301,49.578,159.449
C00841=1021.368,232.850,-125.588,169.297,49.583,159.450
C00842=1021.362,232.602,-125.561,169.293,49.587,159.450
C00843=1021.356,232.353,-125.533,169.290,49.592,159.451
C00844=1021.350,232.105,-125.507,169.286,49.596,159.451
C00845=1021.344,231.856,-125.480,169.282,49.602,159.451
C00846=1021.337,231.608,-125.452,169.278,49.607,159.452
C00847=1021.331,231.359,-125.425,169.274,49.611,159.452
C00848=1021.325,231.111,-125.398,169.271,49.616,159.453
C00849=1021.319,230.862,-125.371,169.266,49.621,159.453
C00850=1021.313,230.614,-125.344,169.263,49.625,159.454
C00851=1021.307,230.366,-125.317,169.259,49.630,159.454
C00852=1021.300,230.117,-125.290,169.255,49.635,159.454
C00853=1021.295,229.869,-125.263,169.252,49.640,159.455
C00854=1021.288,229.620,-125.236,169.247,49.645,159.455
C00855=1021.281,229.372,-125.210,169.244,49.650,159.456
C00856=1021.275,229.123,-125.183,169.240,49.655,159.456
C00857=1021.269,228.875,-125.156,169.236,49.660,159.457
C00858=1021.264,228.626,-125.129,169.232,49.665,159.457
C00859=1021.257,228.377,-125.102,169.229,49.670,159.458
C00860=1021.251,228.130,-125.075,169.224,49.674,159.458
C00861=1021.245,227.880,-125.048,169.221,49.679,159.459
C00862=1021.239,227.632,-125.021,169.218,49.684,159.459
C00863=1021.232,227.384,-124.995,169.214,49.689,159.460
C00864=1021.226,227.135,-124.968,169.210,49.694,159.460
C00865=1021.220,226.887,-124.941,169.206,49.699,159.460
C00866=1021.214,226.638,-124.914,169.202,49.704,159.461
C00867=1021.207,226.390,-124.888,169.198,49.709,159.461
C00868=1021.201,226.142,-124.861,169.195,49.714,159.462
C00869=1021.195,225.893,-124.834,169.191,49.719,159.462
C00870=1021.188,225.645,-124.808,169.188,49.724,159.463
C00871=1021.183,225.396,-124.781,169.183,49.730,159.463
C00872=1021.176,225.147,-124.754,169.180,49.734,159.464
C00873=1021.170,224.899,-124.728,169.176,49.740,159.464
C00874=1021.164,224.649,-124.702,169.173,49.745,159.465
C00875=1021.158,224.401,-124.675,169.168,49.750,159.465
C00876=1021.151,224.153,-124.649,169.164,49.755,159.466
C00877=1021.145,223.904,-124.622,169.161,49.760,159.466
C00878=1021.139,223.656,-124.596,169.157,49.765,159.467
C00879=1021.133,223.408,-124.570,169.153,49.770,159.467
C00880=1021.126,223.159,-124.542,169.149,49.776,159.468
C00881=1021.120,222.911,-124.516,169.146,49.781,159.468
C00882=1021.114,222.662,-124.490,169.142,49.786,159.469
C00883=1021.108,222.414,-124.463,169.139,49.791,159.469
C00884=1021.102,222.164,-124.437,169.135,49.797,159.470
C00885=1021.096,221.916,-124.411,169.131,49.802,159.471
C00886=1021.089,221.668,-124.385,169.127,49.807,159.471
C00887=1021.083,221.419,-124.358,169.124,49.812,159.472
C00888=1021.077,221.171,-124.331,169.120,49.817,159.472
C00889=1021.071,220.923,-124.305,169.117,49.822,159.473
C00890=1021.065,220.674,-124.279,169.112,49.827,159.473
C00891=1021.058,220.425,-124.253,169.109,49.832,159.474
C00892=1021.053,220.205,-124.229,169.106,49.837,159.474
C00893=1021.047,219.985,-124.205,169.103,49.842,159.475
C00894=1021.043,219.765,-124.182,169.099,49.846,159.475
C00895=1021.037,219.544,-124.159,169.096,49.851,159.476
C00896=1021.031,219.323,-124.135,169.092,49.856,159.476
C00897=1021.026,219.103,-124.112,169.089,49.861,159.476
C00898=1021.020,218.883,-124.089,169.086,49.865,159.477
C00899=1021.016,218.663,-124.066,169.083,49.870,159.477
C00900=1021.008,218.414,-124.040,169.079,49.875,159.478
C00901=1021.003,218.166,-124.013,169.075,49.881,159.479
C00902=1020.996,217.917,-123.988,169.072,49.886,159.479
C00903=1020.990,217.669,-123.962,169.068,49.891,159.480
C00904=1020.984,217.420,-123.936,169.065,49.897,159.480
C00905=1020.978,217.172,-123.910,169.061,49.902,159.481
C00906=1020.971,216.923,-123.883,169.057,49.907,159.481
C00907=1020.965,216.674,-123.857,169.054,49.913,159.482
C00908=1020.959,216.426,-123.831,169.050,49.918,159.482
C00909=1020.953,216.178,-123.806,169.047,49.924,159.483
C00910=1020.947,215.929,-123.779,169.042,49.929,159.484
C00911=1020.940,215.680,-123.753,169.038,49.934,159.484
C00912=1020.934,215.432,-123.727,169.035,49.940,159.485
C00913=1020.928,215.183,-123.701,169.031,49.945,159.485
C00914=1020.922,214.935,-123.675,169.028,49.951,159.486
C00915=1020.915,214.686,-123.650,169.024,49.956,159.486
C00916=1020.910,214.437,-123.624,169.020,49.962,159.487
C00917=1020.903,214.188,-123.598,169.017,49.967,159.488
C00918=1020.897,213.940,-123.572,169.013,49.973,159.488
C00919=1020.890,213.692,-123.546,169.010,49.978,159.489
C00920=1020.885,213.443,-123.520,169.006,49.984,159.489
C00921=1020.878,213.195,-123.494,169.002,49.989,159.490
C00922=1020.872,212.946,-123.469,168.999,49.995,159.491
C00923=1020.866,212.697,-123.443,168.995,50.000,159.491
C00924=1020.860,212.449,-123.417,168.992,50.006,159.492
C00925=1020.854,212.200,-123.392,168.988,50.011,159.492
C00926=1020.848,211.952,-123.365,168.984,50.017,159.493
C00927=1020.841,211.702,-123.339,168.981,50.022,159.494
C00928=1020.835,211.454,-123.314,168.977,50.028,159.494
C00929=1020.829,211.205,-123.287,168.974,50.034,159.495
C00930=1020.823,210.957,-123.262,168.970,50.039,159.495
C00931=1020.817,210.708,-123.237,168.966,50.045,159.496
C00932=1020.811,210.460,-123.210,168.963,50.050,159.497
C00933=1020.805,210.211,-123.185,168.959,50.056,159.497
C00934=1020.799,209.962,-123.159,168.956,50.062,159.498
C00935=1020.792,209.714,-123.134,168.952,50.067,159.498
C00936=1020.786,209.466,-123.108,168.948,50.073,159.499
C00937=1020.780,209.217,-123.083,168.946,50.079,159.500
C00938=1020.774,208.968,-123.057,168.941,50.084,159.500
C00939=1020.768,208.719,-123.031,168.937,50.090,159.501
C00940=1020.762,208.471,-123.006,168.935,50.096,159.502
C00941=1020.756,208.222,-122.981,168.931,50.102,159.502
C00942=1020.749,207.974,-122.955,168.927,50.107,159.503
C00943=1020.743,207.725,-122.929,168.924,50.113,159.503
C00944=1020.737,207.477,-122.904,168.920,50.119,159.504
C00945=1020.730,207.228,-122.879,168.916,50.125,159.505
C00946=1020.724,206.979,-122.853,168.913,50.130,159.505
C00947=1020.718,206.731,-122.828,168.909,50.136,159.506
C00948=1020.712,206.482,-122.803,168.905,50.141,159.507
C00949=1020.706,206.233,-122.777,168.903,50.147,159.507
C00950=1020.699,205.985,-122.752,168.899,50.153,159.508
C00951=1020.694,205.736,-122.726,168.895,50.159,159.509
C00952=1020.688,205.519,-122.704,168.892,50.164,159.509
C00953=1020.682,205.300,-122.682,168.889,50.169,159.510
C00954=1020.677,205.083,-122.660,168.885,50.174,159.510
C00955=1020.672,204.865,-122.638,168.883,50.180,159.511
C00956=1020.666,204.647,-122.615,168.879,50.185,159.512
C00957=1020.661,204.430,-122.593,168.876,50.190,159.512
C00958=1020.655,204.212,-122.572,168.873,50.195,159.513
C00959=1020.649,203.994,-122.550,168.870,50.200,159.513
C00960=1020.628,202.955,-122.450,168.425,50.106,159.419
C00961=1020.623,202.706,-122.427,168.421,50.113,159.420
C00962=1020.616,202.458,-122.403,168.416,50.120,159.421
C00963=1020.612,202.208,-122.379,168.411,50.126,159.421
C00964=1020.606,201.960,-122.355,168.407,50.133,159.422
C00965=1020.600,201.711,-122.332,168.402,50.140,159.423
C00966=1020.595,201.462,-122.309,168.399,50.147,159.423
C00967=1020.590,201.213,-122.284,168.394,50.154,159.424
C00968=1020.585,200.964,-122.261,168.389,50.160,159.425
C00969=1020.579,200.716,-122.237,168.385,50.167,159.425
C00970=1020.575,200.467,-122.214,168.381,50.174,159.426
C00971=1020.570,200.218,-122.190,168.377,50.181,159.427
C00972=1020.564,199.969,-122.166,168.372,50.188,159.428
C00973=1020.559,199.720,-122.143,168.368,50.194,159.428
C00974=1020.554,199.471,-122.120,168.363,50.201,159.429
C00975=1020.548,199.222,-122.097,168.360,50.208,159.430
C00976=1020.543,198.973,-122.073,168.355,50.215,159.430
C00977=1020.537,198.725,-122.050,168.351,50.222,159.431
C00978=1020.531,198.476,-122.027,168.346,50.229,159.432
C00979=1020.526,198.227,-122.003,168.342,50.236,159.432
C00980=1020.521,197.979,-121.980,168.337,50.243,159.433
C00981=1020.515,197.730,-121.958,168.334,50.250,159.434
C00982=1020.510,197.480,-121.934,168.329,50.257,159.435
C00983=1020.505,197.232,-121.911,168.325,50.264,159.435
C00984=1020.499,196.983,-121.888,168.320,50.271,159.436
C00985=1020.494,196.733,-121.865,168.316,50.278,159.437
C00986=1020.488,196.485,-121.842,168.311,50.285,159.437
C00987=1020.483,196.236,-121.819,168.308,50.292,159.438
C00988=1020.478,195.987,-121.795,168.303,50.299,159.439
C00989=1020.472,195.738,-121.773,168.299,50.306,159.440
C00990=1020.467,195.489,-121.750,168.294,50.313,159.440
C00991=1020.462,195.240,-121.726,168.291,50.320,159.441
C00992=1020.457,194.992,-121.703,168.287,50.327,159.442
C00993=1020.452,194.743,-121.680,168.282,50.335,159.443
C00994=1020.446,194.494,-121.657,168.278,50.342,159.443
C00995=1020.440,194.245,-121.634,168.274,50.348,159.444
C00996=1020.435,193.996,-121.611,168.270,50.355,159.445
C00997=1020.430,193.748,-121.588,168.265,50.362,159.446
C00998=1020.424,193.499,-121.565,168.261,50.370,159.446
C00999=1020.419,193.249,-121.541,168.257,50.376,159.447
C01000=1020.413,193.001,-121.518,168.253,50.383,159.448
C01001=1020.409,192.752,-121.497,168.248,50.390,159.449
C01002=1020.404,192.502,-121.473,168.244,50.397,159.449
C01003=1020.398,192.254,-121.450,168.241,50.404,159.450
C01004=1020.393,192.005,-121.428,168.236,50.411,159.451
C01005=1020.388,191.756,-121.404,168.232,50.418,159.451
C01006=1020.382,191.507,-121.381,168.228,50.425,159.452
C01007=1020.377,191.258,-121.359,168.224,50.432,159.453
C01008=1020.372,191.010,-121.336,168.219,50.439,159.454
C01009=1020.367,190.760,-121.313,168.216,50.446,159.454
C01010=1020.361,190.511,-121.290,168.211,50.453,159.455
C01011=1020.356,190.263,-121.267,168.207,50.460,159.456
C01012=1020.351,190.013,-121.244,168.203,50.467,159.457
C01013=1020.345,189.765,-121.221,168.199,50.474,159.457
C01014=1020.340,189.516,-121.199,168.194,50.481,159.458
C01015=1020.335,189.267,-121.175,168.191,50.488,159.459
C01016=1020.330,189.018,-121.153,168.187,50.495,159.460
C01017=1020.325,188.769,-121.131,168.182,50.502,159.460
C01018=1020.320,188.520,-121.107,168.179,50.509,159.461
C01019=1020.314,188.272,-121.084,168.175,50.517,159.462
C01020=1020.309,188.023,-121.062,168.170,50.524,159.463
C01021=1020.303,187.741,-121.036,168.166,50.531,159.463
C01022=1020.298,187.460,-121.010,168.161,50.539,159.464
C01023=1020.292,187.179,-120.985,168.157,50.547,159.465
C01024=1020.287,186.898,-120.959,168.153,50.555,159.466
C01025=1020.281,186.648,-120.937,168.148,50.562,159.467
C01026=1020.275,186.399,-120.914,168.144,50.569,159.467
C01027=1020.271,186.151,-120.890,168.141,50.576,159.468
C01028=1020.266,185.901,-120.868,168.136,50.583,159.469
C01029=1020.260,185.653,-120.846,168.133,50.590,159.470
C01030=1020.255,185.403,-120.823,168.128,50.597,159.470
C01031=1020.251,185.155,-120.800,168.124,50.604,159.471
C01032=1020.245,184.906,-120.777,168.120,50.611,159.472
C01033=1020.240,184.657,-120.755,168.116,50.618,159.473
C01034=1020.235,184.408,-120.732,168.113,50.625,159.473
C01035=1020.230,184.159,-120.710,168.108,50.632,159.474
C01036=1020.225,183.910,-120.687,168.105,50.639,159.475
C01037=1020.220,183.661,-120.665,168.100,50.646,159.476
C01038=1020.215,183.412,-120.642,168.097,50.653,159.476
C01039=1020.210,183.164,-120.620,168.092,50.660,159.477
C01040=1020.204,182.915,-120.597,168.089,50.666,159.478
C01041=1020.200,182.665,-120.574,168.085,50.674,159.479
C01042=1020.194,182.417,-120.551,168.082,50.681,159.480
C01043=1020.190,182.167,-120.529,168.077,50.688,159.480
C01044=1020.184,181.918,-120.507,168.073,50.695,159.481
C01045=1020.178,181.669,-120.484,168.069,50.702,159.482
C01046=1020.174,181.421,-120.463,168.065,50.710,159.483
C01047=1020.167,181.171,-120.441,168.061,50.717,159.483
C01048=1020.163,180.923,-120.419,168.057,50.724,159.484
C01049=1020.157,180.673,-120.397,168.053,50.732,159.485
C01050=1020.152,180.425,-120.376,168.049,50.739,159.486
C01051=1020.146,180.175,-120.353,168.046,50.746,159.487
C01052=1020.141,179.927,-120.331,168.041,50.753,159.487
C01053=1020.135,179.678,-120.310,168.038,50.760,159.488
C01054=1020.130,179.429,-120.287,168.034,50.768,159.489
C01055=1020.125,179.180,-120.265,168.030,50.775,159.490
C01056=1020.119,178.931,-120.244,168.026,50.782,159.491
C01057=1020.114,178.682,-120.222,168.022,50.790,159.492
C01058=1020.109,178.432,-120.200,168.018,50.797,159.492
C01059=1020.103,178.184,-120.178,168.015,50.804,159.493
C01060=1020.098,177.934,-120.156,168.010,50.812,159.494
C01061=1020.093,177.686,-120.134,168.007,50.818,159.495
C01062=1020.087,177.437,-120.113,168.003,50.826,159.496
C01063=1020.082,177.188,-120.091,167.999,50.833,159.496
C01064=1020.077,176.939,-120.069,167.995,50.840,159.497
C01065=1020.071,176.690,-120.047,167.991,50.848,159.498
C01066=1020.066,176.441,-120.025,167.988,50.855,159.499
C01067=1020.061,176.192,-120.004,167.984,50.863,159.500
C01068=1020.055,175.943,-119.982,167.979,50.870,159.500
C01069=1020.050,175.694,-119.960,167.976,50.877,159.501
C01070=1020.045,175.444,-119.938,167.972,50.884,159.502
C01071=1020.039,175.196,-119.917,167.969,50.891,159.503
C01072=1020.035,174.947,-119.895,167.964,50.898,159.503
C01073=1020.029,174.698,-119.872,167.961,50.906,159.504
C01074=1020.024,174.449,-119.851,167.957,50.913,159.505
C01075=1020.019,174.200,-119.829,167.954,50.921,159.506
C01076=1020.013,173.951,-119.807,167.949,50.928,159.507
C01077=1020.008,173.702,-119.787,167.946,50.935,159.508
C01078=1020.003,173.453,-119.765,167.942,50.942,159.509
C01079=1019.997,173.204,-119.743,167.939,50.949,159.509
C01080=1019.992,172.955,-119.721,167.934,50.956,159.510
C01081=1019.987,172.706,-119.699,167.930,50.964,159.511
C01082=1019.981,172.457,-119.678,167.927,50.971,159.512
C01083=1019.976,172.208,-119.656,167.923,50.979,159.513
C01084=1019.972,171.958,-119.635,167.920,50.986,159.513
C01085=1019.966,171.677,-119.610,167.916,50.994,159.514
C01086=1019.960,171.395,-119.586,167.911,51.003,159.515
C01087=1019.954,171.114,-119.561,167.907,51.011,159.516
C01088=1019.948,170.832,-119.537,167.903,51.018,159.517
C01089=1019.943,170.583,-119.515,167.899,51.026,159.518
C01090=1019.938,170.333,-119.493,167.896,51.033,159.519
C01091=1019.932,170.085,-119.472,167.891,51.040,159.519
C01092=1019.927,169.836,-119.450,167.888,51.048,159.520
C01093=1019.923,169.587,-119.429,167.884,51.055,159.521
C01094=1019.917,169.337,-119.407,167.881,51.062,159.522
C01095=1019.912,169.089,-119.385,167.877,51.070,159.523
C01096=1019.907,168.839,-119.365,167.873,51.077,159.524
C01097=1019.902,168.591,-119.343,167.870,51.084,159.525
C01098=1019.897,168.342,-119.321,167.866,51.091,159.525
C01099=1019.891,168.093,-119.300,167.862,51.098,159.526
C01100=1019.886,167.843,-119.278,167.859,51.106,159.527
C01101=1019.881,167.594,-119.257,167.855,51.113,159.528
C01102=1019.876,167.346,-119.235,167.852,51.120,159.529
C01103=1019.871,167.096,-119.214,167.848,51.128,159.529
C01104=1019.866,166.848,-119.193,167.845,51.135,159.530
C01105=1019.860,166.598,-119.171,167.840,51.142,159.531
C01106=1019.856,166.349,-119.149,167.837,51.149,159.532
C01107=1019.850,166.101,-119.128,167.834,51.156,159.533
C01108=1019.846,165.851,-119.107,167.829,51.163,159.533
C01109=1019.841,165.602,-119.085,167.827,51.171,159.534
C01110=1019.835,165.354,-119.064,167.822,51.178,159.535
C01111=1019.831,165.104,-119.043,167.819,51.185,159.536
C01112=1019.825,164.856,-119.021,167.816,51.193,159.537
C01113=1019.820,164.606,-119.000,167.812,51.200,159.538
C01114=1019.815,164.357,-118.978,167.808,51.207,159.538
C01115=1019.810,164.108,-118.957,167.805,51.214,159.539
C01116=1019.805,163.859,-118.936,167.801,51.221,159.540
C01117=1019.801,163.610,-118.914,167.798,51.228,159.541
C01118=1019.795,163.361,-118.893,167.795,51.236,159.542
C01119=1019.790,163.112,-118.871,167.790,51.243,159.542
C01120=1019.785,162.863,-118.851,167.787,51.250,159.543
C01121=1019.780,162.614,-118.829,167.784,51.258,159.544
C01122=1019.776,162.365,-118.808,167.780,51.265,159.545
C01123=1019.770,162.116,-118.787,167.776,51.272,159.546
C01124=1019.766,161.867,-118.765,167.773,51.279,159.547
C01125=1019.760,161.618,-118.744,167.769,51.286,159.547
C01126=1019.755,161.368,-118.723,167.766,51.293,159.548
C01127=1019.750,161.119,-118.701,167.763,51.301,159.549
C01128=1019.745,160.870,-118.680,167.760,51.308,159.550
C01129=1019.740,160.621,-118.658,167.755,51.315,159.551
C01130=1019.736,160.372,-118.637,167.752,51.323,159.552
C01131=1019.730,160.124,-118.616,167.749,51.330,159.552
C01132=1019.726,159.874,-118.595,167.745,51.337,159.553
C01133=1019.720,159.625,-118.574,167.741,51.344,159.554
C01134=1019.715,159.376,-118.552,167.738,51.351,159.555
C01135=1019.711,159.127,-118.531,167.735,51.358,159.556
C01136=1019.705,158.878,-118.510,167.731,51.365,159.556
C01137=1019.701,158.629,-118.489,167.728,51.373,159.557
C01138=1019.696,158.380,-118.468,167.725,51.380,159.558
C01139=1019.690,158.131,-118.448,167.721,51.388,159.559
C01140=1019.685,157.881,-118.427,167.717,51.395,159.560
C01141=1019.680,157.633,-118.406,167.714,51.402,159.561
C01142=1019.674,157.384,-118.385,167.710,51.410,159.562
C01143=1019.669,157.135,-118.365,167.707,51.417,159.563
C01144=1019.665,156.885,-118.344,167.704,51.425,159.564
C01145=1019.659,156.636,-118.323,167.700,51.432,159.564
C01146=1019.654,156.387,-118.303,167.697,51.440,159.565
C01147=1019.649,156.138,-118.282,167.693,51.447,159.566
C01148=1019.643,155.889,-118.261,167.690,51.454,159.567
C01149=1019.638,155.607,-118.238,167.686,51.462,159.568
C01150=1019.632,155.325,-118.214,167.682,51.471,159.569
C01151=1019.626,155.043,-118.191,167.679,51.479,159.570
C01152=1019.620,154.761,-118.167,167.674,51.488,159.571
C01153=1019.615,154.512,-118.147,167.671,51.495,159.572
C01154=1019.610,154.263,-118.126,167.668,51.503,159.573
C01155=1019.605,154.014,-118.105,167.665,51.510,159.573
C01156=1019.599,153.765,-118.085,167.661,51.517,159.574
C01157=1019.595,153.515,-118.064,167.657,51.524,159.575
C01158=1019.590,153.266,-118.043,167.655,51.532,159.576
C01159=1019.584,153.017,-118.023,167.650,51.539,159.577
C01160=1019.580,152.769,-118.003,167.647,51.547,159.578
C01161=1019.574,152.519,-117.982,167.644,51.554,159.579
C01162=1019.569,152.270,-117.961,167.640,51.562,159.579
C01163=1019.564,152.021,-117.941,167.637,51.569,159.580
C01164=1019.559,151.772,-117.920,167.634,51.576,159.581
C01165=1019.553,151.523,-117.900,167.630,51.584,159.582
C01166=1019.548,151.273,-117.880,167.627,51.591,159.583
C01167=1019.543,151.024,-117.859,167.624,51.599,159.584
C01168=1019.538,150.775,-117.839,167.620,51.606,159.585
C01169=1019.533,150.526,-117.818,167.617,51.614,159.586
C01170=1019.528,150.277,-117.798,167.614,51.621,159.587
C01171=1019.523,150.028,-117.777,167.611,51.628,159.587
C01172=1019.518,149.779,-117.757,167.607,51.636,159.588
C01173=1019.512,149.530,-117.736,167.604,51.643,159.589
C01174=1019.507,149.280,-117.717,167.601,51.651,159.590
C01175=1019.502,149.031,-117.696,167.596,51.658,159.591
C01176=1019.497,148.782,-117.675,167.594,51.666,159.592
C01177=1019.492,148.534,-117.655,167.590,51.673,159.593
C01178=1019.487,148.284,-117.635,167.587,51.680,159.594
C01179=1019.481,148.035,-117.615,167.584,51.688,159.594
C01180=1019.476,147.786,-117.595,167.580,51.695,159.595
C01181=1019.471,147.537,-117.574,167.577,51.703,159.596
C01182=1019.465,147.288,-117.554,167.574,51.710,159.597
C01183=1019.461,147.039,-117.534,167.570,51.718,159.598
C01184=1019.456,146.789,-117.514,167.567,51.725,159.599
C01185=1019.451,146.540,-117.493,167.564,51.733,159.600
C01186=1019.445,146.291,-117.473,167.561,51.740,159.601
C01187=1019.440,146.041,-117.453,167.557,51.748,159.601
C01188=1019.436,145.793,-117.433,167.554,51.755,159.602
C01189=1019.430,145.544,-117.413,167.551,51.762,159.603
C01190=1019.425,145.294,-117.393,167.547,51.770,159.604
C01191=1019.420,145.045,-117.372,167.544,51.778,159.605
C01192=1019.415,144.796,-117.352,167.541,51.785,159.606
C01193=1019.409,144.548,-117.333,167.538,51.792,159.607
C01194=1019.404,144.298,-117.312,167.534,51.801,159.608
C01195=1019.399,144.049,-117.292,167.531,51.807,159.608
C01196=1019.393,143.800,-117.273,167.528,51.815,159.610
C01197=1019.389,143.551,-117.253,167.524,51.823,159.610
C01198=1019.383,143.302,-117.232,167.521,51.830,159.611
C01199=1019.378,143.052,-117.213,167.518,51.838,159.612
C01200=1019.372,142.803,-117.193,167.516,51.845,159.613
C01201=1019.368,142.554,-117.173,167.511,51.853,159.614
C01202=1019.363,142.305,-117.153,167.509,51.860,159.615
C01203=1019.357,142.056,-117.133,167.505,51.867,159.616
C01204=1019.352,141.806,-117.113,167.502,51.875,159.617
C01205=1019.348,141.557,-117.093,167.499,51.883,159.618
C01206=1019.342,141.309,-117.073,167.495,51.890,159.618
C01207=1019.337,141.059,-117.054,167.493,51.898,159.619
C01208=1019.331,140.810,-117.033,167.490,51.905,159.620
C01209=1019.326,140.561,-117.014,167.487,51.912,159.621
C01210=1019.321,140.312,-116.994,167.483,51.920,159.622
C01211=1019.316,140.062,-116.974,167.479,51.927,159.623
C01212=1019.311,139.814,-116.954,167.477,51.935,159.624
C01213=1019.305,139.531,-116.932,167.473,51.944,159.625
C01214=1019.300,139.249,-116.909,167.469,51.952,159.626
C01215=1019.294,138.967,-116.887,167.466,51.961,159.627
C01216=1019.287,138.684,-116.864,167.462,51.969,159.628
C01217=1019.283,138.435,-116.844,167.459,51.976,159.629
C01218=1019.278,138.186,-116.824,167.456,51.984,159.630
C01219=1019.272,137.937,-116.805,167.452,51.991,159.630
C01220=1019.268,137.688,-116.785,167.450,51.999,159.631
C01221=1019.262,137.439,-116.765,167.447,52.007,159.632
C01222=1019.257,137.189,-116.745,167.443,52.014,159.633
C01223=1019.252,136.941,-116.727,167.440,52.022,159.634
C01224=1019.247,136.691,-116.707,167.437,52.030,159.635
C01225=1019.241,136.442,-116.687,167.434,52.037,159.636
C01226=1019.236,136.193,-116.667,167.431,52.044,159.637
C01227=1019.231,135.944,-116.648,167.427,52.052,159.638
C01228=1019.226,135.694,-116.629,167.424,52.059,159.639
C01229=1019.220,135.446,-116.609,167.421,52.067,159.640
C01230=1019.215,135.196,-116.589,167.418,52.075,159.641
C01231=1019.210,134.947,-116.570,167.415,52.082,159.641
C01232=1019.205,134.697,-116.550,167.411,52.090,159.642
C01233=1019.200,134.448,-116.531,167.409,52.098,159.643
C01234=1019.195,134.200,-116.511,167.406,52.105,159.644
C01235=1019.189,133.950,-116.491,167.403,52.112,159.645
C01236=1019.185,133.701,-116.472,167.399,52.120,159.646
C01237=1019.179,133.452,-116.453,167.396,52.128,159.647
C01238=1019.174,133.202,-116.433,167.393,52.135,159.648
C01239=1019.169,132.953,-116.414,167.390,52.143,159.649
C01240=1019.163,132.704,-116.394,167.387,52.151,159.650
C01241=1019.159,132.455,-116.375,167.383,52.158,159.650
C01242=1019.153,132.206,-116.355,167.380,52.166,159.652
C01243=1019.149,131.957,-116.336,167.378,52.173,159.653
C01244=1019.143,131.707,-116.317,167.374,52.180,159.653
C01245=1019.137,131.458,-116.297,167.372,52.188,159.654
C01246=1019.133,131.209,-116.278,167.369,52.196,159.655
C01247=1019.127,130.960,-116.259,167.365,52.203,159.656
C01248=1019.123,130.710,-116.239,167.362,52.211,159.657
C01249=1019.117,130.461,-116.220,167.359,52.219,159.658
C01250=1019.113,130.212,-116.200,167.356,52.226,159.659
C01251=1019.107,129.963,-116.181,167.353,52.233,159.660
C01252=1019.102,129.713,-116.162,167.351,52.241,159.661
C01253=1019.097,129.464,-116.143,167.346,52.249,159.661
C01254=1019.092,129.215,-116.123,167.344,52.256,159.662
C01255=1019.087,128.966,-116.104,167.341,52.264,159.664
C01256=1019.081,128.717,-116.085,167.338,52.272,159.665
C01257=1019.076,128.468,-116.066,167.334,52.280,159.665
C01258=1019.070,128.218,-116.047,167.332,52.288,159.666
C01259=1019.065,127.969,-116.029,167.328,52.295,159.667
C01260=1019.060,127.720,-116.010,167.326,52.302,159.668
C01261=1019.054,127.471,-115.991,167.322,52.310,159.669
C01262=1019.049,127.221,-115.971,167.319,52.318,159.670
C01263=1019.044,126.973,-115.953,167.316,52.326,159.671
C01264=1019.038,126.723,-115.933,167.313,52.333,159.672
C01265=1019.033,126.474,-115.915,167.311,52.341,159.673
C01266=1019.028,126.224,-115.896,167.307,52.349,159.674
C01267=1019.023,125.975,-115.876,167.304,52.357,159.675
C01268=1019.018,125.726,-115.857,167.301,52.364,159.676
C01269=1019.012,125.477,-115.838,167.298,52.371,159.677
C01270=1019.007,125.227,-115.820,167.294,52.380,159.678
C01271=1019.002,124.978,-115.801,167.292,52.387,159.679
C01272=1018.996,124.729,-115.782,167.289,52.395,159.680
C01273=1018.991,124.480,-115.763,167.286,52.402,159.680
C01274=1018.986,124.230,-115.744,167.283,52.410,159.681
C01275=1018.981,123.982,-115.725,167.280,52.418,159.682
C01276=1018.975,123.732,-115.706,167.277,52.426,159.683
C01277=1018.970,123.450,-115.685,167.273,52.435,159.684
C01278=1018.964,123.168,-115.664,167.270,52.443,159.685
C01279=1018.958,122.885,-115.642,167.266,52.452,159.686
C01280=1018.952,122.603,-115.621,167.263,52.460,159.687
C01281=1018.946,122.354,-115.602,167.260,52.468,159.688
C01282=1018.941,122.104,-115.583,167.257,52.475,159.689
C01283=1018.936,121.856,-115.564,167.254,52.483,159.690
C01284=1018.931,121.607,-115.545,167.252,52.491,159.691
C01285=1018.926,121.357,-115.527,167.249,52.499,159.692
C01286=1018.920,121.108,-115.508,167.245,52.506,159.693
C01287=1018.915,120.858,-115.488,167.242,52.514,159.694
C01288=1018.911,120.609,-115.470,167.239,52.521,159.695
C01289=1018.906,120.360,-115.451,167.236,52.529,159.696
C01290=1018.900,120.111,-115.432,167.234,52.536,159.697
C01291=1018.895,119.861,-115.414,167.231,52.544,159.698
C01292=1018.889,119.612,-115.395,167.228,52.552,159.699
C01293=1018.884,119.363,-115.376,167.225,52.559,159.700
C01294=1018.880,119.114,-115.357,167.221,52.567,159.700
C01295=1018.874,118.864,-115.338,167.219,52.575,159.701
C01296=1018.869,118.615,-115.320,167.216,52.582,159.702
C01297=1018.864,118.366,-115.301,167.213,52.590,159.703
C01298=1018.858,118.117,-115.282,167.210,52.598,159.704
C01299=1018.854,117.868,-115.264,167.207,52.605,159.705
C01300=1018.848,117.619,-115.245,167.204,52.612,159.706
C01301=1018.843,117.369,-115.226,167.202,52.620,159.707
C01302=1018.838,117.120,-115.208,167.199,52.627,159.708
C01303=1018.833,116.871,-115.189,167.196,52.635,159.709
C01304=1018.828,116.621,-115.170,167.192,52.643,159.710
C01305=1018.823,116.372,-115.151,167.189,52.650,159.711
C01306=1018.818,116.123,-115.132,167.186,52.658,159.712
C01307=1018.813,115.873,-115.113,167.184,52.666,159.713
C01308=1018.808,115.624,-115.095,167.181,52.673,159.713
C01309=1018.803,115.375,-115.076,167.178,52.681,159.714
C01310=1018.797,115.125,-115.058,167.175,52.689,159.715
C01311=1018.792,114.877,-115.039,167.172,52.696,159.716
C01312=1018.788,114.627,-115.021,167.170,52.704,159.717
C01313=1018.783,114.379,-115.002,167.167,52.711,159.718
C01314=1018.777,114.128,-114.983,167.164,52.719,159.719
C01315=1018.772,113.880,-114.964,167.161,52.726,159.720
C01316=1018.767,113.630,-114.946,167.158,52.733,159.721
C01317=1018.762,113.382,-114.927,167.155,52.741,159.722
C01318=1018.757,113.132,-114.909,167.153,52.749,159.723
C01319=1018.752,112.883,-114.890,167.150,52.756,159.724
C01320=1018.747,112.634,-114.872,167.147,52.764,159.725
C01321=1018.742,112.383,-114.853,167.144,52.771,159.726
C01322=1018.736,112.135,-114.834,167.141,52.779,159.727
C01323=1018.732,111.885,-114.816,167.138,52.787,159.727
C01324=1018.727,111.636,-114.798,167.135,52.795,159.728
C01325=1018.721,111.387,-114.779,167.132,52.802,159.729
C01326=1018.716,111.138,-114.761,167.129,52.810,159.730
C01327=1018.711,110.888,-114.743,167.127,52.818,159.731
C01328=1018.706,110.640,-114.724,167.124,52.825,159.732
C01329=1018.700,110.389,-114.706,167.121,52.833,159.733
C01330=1018.695,110.140,-114.688,167.118,52.840,159.734
C01331=1018.690,109.891,-114.670,167.116,52.848,159.735
C01332=1018.685,109.642,-114.651,167.111,52.856,159.736
C01333=1018.680,109.392,-114.633,167.109,52.864,159.737
C01334=1018.674,109.143,-114.615,167.106,52.871,159.738
C01335=1018.669,108.894,-114.597,167.104,52.879,159.739
C01336=1018.664,108.645,-114.579,167.101,52.887,159.740
C01337=1018.659,108.395,-114.561,167.098,52.895,159.741
C01338=1018.653,108.146,-114.542,167.095,52.902,159.742
C01339=1018.648,107.897,-114.524,167.092,52.910,159.743
C01340=1018.643,107.648,-114.506,167.089,52.918,159.744
C01341=1018.638,107.426,-114.490,167.087,52.925,159.745
C01342=1018.634,107.204,-114.475,167.084,52.932,159.745
C01343=1018.629,106.982,-114.458,167.082,52.939,159.746
C01344=1018.624,106.761,-114.442,167.079,52.946,159.747
C01345=1018.619,106.538,-114.427,167.077,52.953,159.748
C01346=1018.614,106.316,-114.410,167.075,52.959,159.749
C01347=1018.610,106.095,-114.394,167.071,52.966,159.749
C01348=1018.605,105.873,-114.377,167.069,52.973,159.750
C01349=1018.598,105.536,-114.354,167.065,52.984,159.752
C01350=1018.591,105.199,-114.329,167.061,52.994,159.753
C01351=1018.584,104.862,-114.305,167.058,53.004,159.754
C01352=1018.578,104.525,-114.280,167.054,53.014,159.756
C01353=1018.571,104.275,-114.262,167.051,53.022,159.757
C01354=1018.567,104.025,-114.244,167.048,53.030,159.757
C01355=1018.561,103.776,-114.227,167.045,53.038,159.758
C01356=1018.556,103.527,-114.208,167.042,53.045,159.759
C01357=1018.551,103.278,-114.191,167.039,53.053,159.760
C01358=1018.546,103.029,-114.173,167.037,53.061,159.761
C01359=1018.541,102.780,-114.155,167.034,53.069,159.762
C01360=1018.536,102.530,-114.137,167.031,53.076,159.763
C01361=1018.530,102.280,-114.118,167.029,53.084,159.764
C01362=1018.525,102.031,-114.101,167.026,53.092,159.765
C01363=1018.520,101.782,-114.083,167.023,53.099,159.766
C01364=1018.515,101.533,-114.065,167.020,53.107,159.767
C01365=1018.510,101.283,-114.047,167.018,53.115,159.768
C01366=1018.504,101.034,-114.029,167.015,53.123,159.769
C01367=1018.499,100.785,-114.011,167.012,53.130,159.770
C01368=1018.494,100.535,-113.994,167.010,53.138,159.771
C01369=1018.490,100.286,-113.976,167.006,53.146,159.772
C01370=1018.485,100.037,-113.958,167.003,53.153,159.773
C01371=1018.479,99.787,-113.940,167.000,53.161,159.774
C01372=1018.474,99.538,-113.922,166.998,53.169,159.775
C01373=1018.468,99.289,-113.904,166.995,53.176,159.775
C01374=1018.464,99.039,-113.886,166.992,53.184,159.776
C01375=1018.458,98.790,-113.869,166.990,53.192,159.777
C01376=1018.453,98.540,-113.852,166.987,53.200,159.778
C01377=1018.447,98.291,-113.834,166.984,53.208,159.779
C01378=1018.442,98.042,-113.816,166.981,53.215,159.780
C01379=1018.437,97.793,-113.799,166.979,53.223,159.781
C01380=1018.432,97.543,-113.782,166.975,53.231,159.782
C01381=1018.427,97.294,-113.764,166.973,53.239,159.783
C01382=1018.421,97.045,-113.746,166.970,53.247,159.784
C01383=1018.416,96.796,-113.728,166.967,53.254,159.785
C01384=1018.411,96.546,-113.712,166.965,53.262,159.786
C01385=1018.405,96.296,-113.693,166.962,53.270,159.787
C01386=1018.400,96.047,-113.675,166.959,53.277,159.788
C01387=1018.395,95.798,-113.659,166.957,53.285,159.789
C01388=1018.389,95.548,-113.641,166.954,53.293,159.790
C01389=1018.384,95.299,-113.623,166.951,53.300,159.791
C01390=1018.379,95.050,-113.605,166.948,53.309,159.792
C01391=1018.374,94.800,-113.588,166.945,53.317,159.793
C01392=1018.368,94.551,-113.571,166.942,53.324,159.794
C01393=1018.363,94.302,-113.553,166.940,53.332,159.795
C01394=1018.358,94.052,-113.536,166.937,53.340,159.796
C01395=1018.353,93.803,-113.518,166.935,53.348,159.797
C01396=1018.347,93.554,-113.501,166.932,53.355,159.798
C01397=1018.343,93.304,-113.483,166.929,53.363,159.799
C01398=1018.337,93.055,-113.466,166.926,53.371,159.800
C01399=1018.332,92.806,-113.449,166.924,53.378,159.801
C01400=1018.326,92.557,-113.431,166.921,53.386,159.801
C01401=1018.322,92.307,-113.413,166.918,53.394,159.802
C01402=1018.316,92.058,-113.396,166.916,53.401,159.804
C01403=1018.311,91.809,-113.379,166.912,53.410,159.804
C01404=1018.306,91.560,-113.362,166.909,53.417,159.805
C01405=1018.300,91.277,-113.342,166.907,53.426,159.806
C01406=1018.294,90.995,-113.322,166.904,53.435,159.808
C01407=1018.289,90.713,-113.302,166.901,53.443,159.808
C01408=1018.282,90.431,-113.283,166.897,53.452,159.810
C01409=1018.277,90.181,-113.266,166.895,53.460,159.811
C01410=1018.273,89.932,-113.248,166.892,53.467,159.811
C01411=1018.267,89.683,-113.230,166.889,53.475,159.812
C01412=1018.262,89.434,-113.214,166.887,53.483,159.813
C01413=1018.257,89.185,-113.196,166.884,53.490,159.814
C01414=1018.252,88.935,-113.179,166.881,53.498,159.815
C01415=1018.247,88.686,-113.161,166.879,53.506,159.816
C01416=1018.241,88.436,-113.144,166.876,53.514,159.817
C01417=1018.235,88.187,-113.128,166.873,53.522,159.818
C01418=1018.230,87.938,-113.110,166.870,53.530,159.819
C01419=1018.225,87.688,-113.094,166.867,53.537,159.820
C01420=1018.219,87.438,-113.077,166.865,53.545,159.821
C01421=1018.214,87.189,-113.059,166.862,53.553,159.822
C01422=1018.209,86.940,-113.042,166.860,53.561,159.823
C01423=1018.203,86.690,-113.025,166.857,53.569,159.824
C01424=1018.198,86.441,-113.008,166.854,53.576,159.825
C01425=1018.193,86.192,-112.991,166.851,53.585,159.826
C01426=1018.188,85.942,-112.974,166.848,53.592,159.827
C01427=1018.183,85.693,-112.957,166.846,53.600,159.828
C01428=1018.177,85.444,-112.940,166.843,53.608,159.829
C01429=1018.172,85.194,-112.923,166.840,53.616,159.830
C01430=1018.167,84.945,-112.906,166.838,53.624,159.831
C01431=1018.161,84.695,-112.889,166.835,53.631,159.832
C01432=1018.156,84.446,-112.873,166.833,53.639,159.833
C01433=1018.151,84.198,-112.855,166.830,53.647,159.834
C01434=1018.145,83.948,-112.838,166.827,53.655,159.835
C01435=1018.140,83.698,-112.822,166.825,53.663,159.836
C01436=1018.135,83.449,-112.805,166.821,53.671,159.837
C01437=1018.129,83.200,-112.787,166.819,53.679,159.838
C01438=1018.124,82.950,-112.770,166.816,53.686,159.839
C01439=1018.119,82.700,-112.754,166.814,53.694,159.840
C01440=1018.114,82.451,-112.737,166.811,53.702,159.841
C01441=1018.109,82.202,-112.719,166.809,53.710,159.842
C01442=1018.104,81.953,-112.703,166.806,53.717,159.842
C01443=1018.098,81.703,-112.686,166.803,53.725,159.843
C01444=1018.093,81.453,-112.669,166.801,53.733,159.844
C01445=1018.088,81.204,-112.651,166.798,53.740,159.845
C01446=1018.082,80.956,-112.635,166.795,53.748,159.846
C01447=1018.077,80.706,-112.619,166.793,53.756,159.847
C01448=1018.072,80.456,-112.602,166.790,53.763,159.848
C01449=1018.067,80.207,-112.585,166.787,53.771,159.849
C01450=1018.061,79.958,-112.567,166.785,53.779,159.850
C01451=1018.057,79.709,-112.551,166.783,53.787,159.851
C01452=1018.051,79.459,-112.534,166.780,53.795,159.852
C01453=1018.046,79.209,-112.517,166.776,53.803,159.853
C01454=1018.041,78.960,-112.500,166.773,53.810,159.854
C01455=1018.036,78.711,-112.484,166.771,53.818,159.855
C01456=1018.031,78.462,-112.466,166.768,53.826,159.856
C01457=1018.026,78.212,-112.449,166.765,53.833,159.857
C01458=1018.020,77.963,-112.433,166.763,53.841,159.858
C01459=1018.014,77.713,-112.416,166.760,53.849,159.859
C01460=1018.010,77.464,-112.400,166.758,53.857,159.860
C01461=1018.005,77.214,-112.383,166.755,53.865,159.861
C01462=1017.999,76.965,-112.366,166.753,53.873,159.862
C01463=1017.994,76.715,-112.349,166.750,53.880,159.862
C01464=1017.989,76.466,-112.333,166.747,53.888,159.863
C01465=1017.984,76.217,-112.317,166.745,53.896,159.864
C01466=1017.978,75.967,-112.300,166.742,53.904,159.866
C01467=1017.973,75.717,-112.283,166.740,53.911,159.866
C01468=1017.968,75.469,-112.267,166.737,53.919,159.867
C01469=1017.962,75.186,-112.248,166.734,53.928,159.869
C01470=1017.956,74.904,-112.229,166.731,53.937,159.870
C01471=1017.949,74.623,-112.211,166.728,53.946,159.871
C01472=1017.944,74.340,-112.192,166.725,53.955,159.872
C01473=1017.939,74.091,-112.175,166.722,53.963,159.873
C01474=1017.933,73.841,-112.159,166.720,53.971,159.874
C01475=1017.928,73.592,-112.142,166.717,53.978,159.875
C01476=1017.923,73.343,-112.126,166.714,53.986,159.876
C01477=1017.917,73.093,-112.109,166.712,53.994,159.877
C01478=1017.913,72.844,-112.094,166.710,54.002,159.878
C01479=1017.907,72.594,-112.077,166.707,54.009,159.878
C01480=1017.901,72.345,-112.060,166.703,54.018,159.879
C01481=1017.897,72.096,-112.044,166.701,54.026,159.880
C01482=1017.891,71.847,-112.028,166.698,54.033,159.881
C01483=1017.886,71.597,-112.011,166.696,54.041,159.882
C01484=1017.880,71.347,-111.994,166.693,54.049,159.883
C01485=1017.875,71.099,-111.978,166.690,54.056,159.884
C01486=1017.870,70.848,-111.962,166.688,54.064,159.885
C01487=1017.864,70.599,-111.946,166.685,54.072,159.886
C01488=1017.860,70.350,-111.929,166.683,54.080,159.887
C01489=1017.854,70.100,-111.912,166.680,54.088,159.888
C01490=1017.848,69.851,-111.896,166.678,54.096,159.889
C01491=1017.844,69.601,-111.880,166.675,54.104,159.890
C01492=1017.838,69.352,-111.864,166.672,54.111,159.891
C01493=1017.834,69.103,-111.848,166.670,54.119,159.892
C01494=1017.828,68.853,-111.831,166.668,54.127,159.893
C01495=1017.822,68.604,-111.814,166.665,54.134,159.894
C01496=1017.818,68.355,-111.799,166.661,54.143,159.895
C01497=1017.812,68.105,-111.782,166.659,54.151,159.896
C01498=1017.807,67.856,-111.766,166.656,54.158,159.897
C01499=1017.802,67.606,-111.750,166.654,54.166,159.898
C01500=1017.797,67.357,-111.734,166.651,54.174,159.899
C01501=1017.791,67.107,-111.717,166.648,54.181,159.899
C01502=1017.786,66.858,-111.702,166.646,54.189,159.901
C01503=1017.780,66.608,-111.685,166.644,54.197,159.902
C01504=1017.775,66.360,-111.669,166.641,54.205,159.903
C01505=1017.770,66.109,-111.653,166.638,54.213,159.903
C01506=1017.764,65.860,-111.637,166.636,54.221,159.904
C01507=1017.760,65.611,-111.621,166.634,54.229,159.906
C01508=1017.754,65.361,-111.605,166.630,54.236,159.906
C01509=1017.749,65.112,-111.589,166.627,54.244,159.907
C01510=1017.743,64.863,-111.572,166.625,54.252,159.908
C01511=1017.738,64.613,-111.557,166.622,54.260,159.909
C01512=1017.733,64.364,-111.540,166.620,54.268,159.910
C01513=1017.728,64.114,-111.525,166.617,54.276,159.911
C01514=1017.722,63.865,-111.509,166.615,54.284,159.912
C01515=1017.717,63.615,-111.493,166.612,54.291,159.913
C01516=1017.712,63.366,-111.477,166.610,54.299,159.914
C01517=1017.706,63.117,-111.461,166.608,54.307,159.915
C01518=1017.701,62.867,-111.444,166.605,54.315,159.916
C01519=1017.696,62.617,-111.429,166.601,54.323,159.917
C01520=1017.690,62.368,-111.413,166.599,54.331,159.918
C01521=1017.685,62.119,-111.398,166.597,54.339,159.919
C01522=1017.679,61.869,-111.382,166.594,54.347,159.920
C01523=1017.673,61.620,-111.366,166.591,54.355,159.921
C01524=1017.668,61.370,-111.351,166.588,54.363,159.922
C01525=1017.663,61.121,-111.334,166.586,54.371,159.923
C01526=1017.658,60.871,-111.319,166.583,54.379,159.924
C01527=1017.652,60.622,-111.303,166.581,54.387,159.925
C01528=1017.647,60.373,-111.287,166.578,54.394,159.926
C01529=1017.641,60.123,-111.272,166.576,54.403,159.927
C01530=1017.636,59.874,-111.256,166.572,54.411,159.928
C01531=1017.630,59.624,-111.240,166.570,54.419,159.929
C01532=1017.625,59.375,-111.225,166.568,54.427,159.930
C01533=1017.619,59.093,-111.207,166.564,54.436,159.931
C01534=1017.613,58.811,-111.190,166.561,54.445,159.932
C01535=1017.607,58.529,-111.172,166.559,54.454,159.933
C01536=1017.601,58.246,-111.155,166.556,54.463,159.934
C01537=1017.595,57.997,-111.138,166.553,54.471,159.935
C01538=1017.590,57.748,-111.123,166.551,54.478,159.936
C01539=1017.585,57.497,-111.107,166.548,54.486,159.937
C01540=1017.580,57.248,-111.092,166.546,54.495,159.938
C01541=1017.574,56.999,-111.076,166.543,54.503,159.939
C01542=1017.569,56.750,-111.060,166.540,54.510,159.940
C01543=1017.564,56.500,-111.045,166.537,54.518,159.941
C01544=1017.558,56.250,-111.030,166.535,54.527,159.942
C01545=1017.553,56.002,-111.014,166.532,54.534,159.943
C01546=1017.547,55.752,-110.998,166.530,54.542,159.944
C01547=1017.542,55.502,-110.983,166.528,54.550,159.945
C01548=1017.536,55.252,-110.968,166.524,54.558,159.946
C01549=1017.531,55.004,-110.952,166.522,54.566,159.947
C01550=1017.525,54.754,-110.936,166.519,54.574,159.948
C01551=1017.520,54.505,-110.921,166.517,54.582,159.949
C01552=1017.515,54.255,-110.905,166.514,54.589,159.949
C01553=1017.509,54.006,-110.890,166.512,54.597,159.951
C01554=1017.504,53.757,-110.874,166.509,54.606,159.952
C01555=1017.499,53.506,-110.858,166.507,54.613,159.952
C01556=1017.494,53.257,-110.843,166.504,54.621,159.953
C01557=1017.489,53.007,-110.827,166.501,54.629,159.954
C01558=1017.483,52.759,-110.812,166.498,54.637,159.955
C01559=1017.478,52.509,-110.796,166.496,54.645,159.956
C01560=1017.473,52.259,-110.781,166.493,54.652,159.957
C01561=1017.468,52.010,-110.766,166.491,54.660,159.958
C01562=1017.462,51.760,-110.750,166.489,54.668,159.959
C01563=1017.457,51.511,-110.735,166.486,54.676,159.960
C01564=1017.452,51.262,-110.720,166.484,54.684,159.961
C01565=1017.446,51.012,-110.704,166.481,54.691,159.962
C01566=1017.441,50.763,-110.688,166.478,54.699,159.963
C01567=1017.435,50.513,-110.673,166.476,54.708,159.964
C01568=1017.430,50.264,-110.658,166.472,54.715,159.965
C01569=1017.425,50.014,-110.642,166.470,54.723,159.966
C01570=1017.419,49.764,-110.627,166.467,54.731,159.966
C01571=1017.414,49.515,-110.612,166.465,54.739,159.968
C01572=1017.409,49.266,-110.597,166.462,54.746,159.968
C01573=1017.403,49.017,-110.580,166.460,54.754,159.969
C01574=1017.398,48.767,-110.565,166.457,54.762,159.970
C01575=1017.394,48.518,-110.549,166.455,54.770,159.971
C01576=1017.388,48.268,-110.534,166.453,54.778,159.972
C01577=1017.383,48.018,-110.519,166.450,54.785,159.973
C01578=1017.378,47.769,-110.504,166.448,54.793,159.974
C01579=1017.373,47.519,-110.488,166.445,54.801,159.975
C01580=1017.368,47.270,-110.473,166.443,54.809,159.976
C01581=1017.363,47.021,-110.458,166.440,54.816,159.977
C01582=1017.357,46.771,-110.442,166.438,54.824,159.978
C01583=1017.352,46.521,-110.427,166.435,54.832,159.979
C01584=1017.347,46.272,-110.412,166.432,54.839,159.980
C01585=1017.341,46.022,-110.396,166.430,54.847,159.981
C01586=1017.336,45.773,-110.381,166.427,54.855,159.981
C01587=1017.331,45.524,-110.366,166.425,54.863,159.983
C01588=1017.326,45.274,-110.351,166.422,54.870,159.983
C01589=1017.320,45.024,-110.335,166.420,54.878,159.984
C01590=1017.315,44.775,-110.320,166.416,54.886,159.985
C01591=1017.310,44.526,-110.305,166.414,54.894,159.986
C01592=1017.305,44.276,-110.289,166.411,54.902,159.987
C01593=1017.300,44.027,-110.274,166.408,54.909,159.988
C01594=1017.295,43.777,-110.259,166.406,54.917,159.989
C01595=1017.290,43.528,-110.244,166.403,54.925,159.990
C01596=1017.284,43.278,-110.228,166.401,54.933,159.991
C01597=1017.278,42.996,-110.211,166.399,54.941,159.992
C01598=1017.272,42.714,-110.194,166.396,54.949,159.993
C01599=1017.267,42.431,-110.176,166.393,54.959,159.994
C01600=1017.261,42.150,-110.160,166.389,54.967,159.995
C01601=1017.255,41.900,-110.144,166.387,54.975,159.996
C01602=1017.250,41.651,-110.129,166.385,54.983,159.997
C01603=1017.245,41.401,-110.114,166.382,54.991,159.998
C01604=1017.240,41.152,-110.100,166.380,54.998,159.999
C01605=1017.234,40.902,-110.084,166.377,55.006,160.000
C01606=1017.229,40.652,-110.069,166.375,55.014,160.000
C01607=1017.224,40.403,-110.054,166.372,55.022,160.002
C01608=1017.218,40.154,-110.040,166.369,55.030,160.002
C01609=1017.213,39.904,-110.025,166.366,55.038,160.003
C01610=1017.208,39.654,-110.010,166.364,55.045,160.004
C01611=1017.203,39.405,-109.994,166.361,55.054,160.005
C01612=1017.197,39.156,-109.980,166.359,55.061,160.006
C01613=1017.192,38.906,-109.965,166.357,55.069,160.007
C01614=1017.187,38.657,-109.950,166.354,55.077,160.008
C01615=1017.182,38.407,-109.935,166.352,55.085,160.009
C01616=1017.176,38.158,-109.921,166.349,55.092,160.010
C01617=1017.171,37.908,-109.906,166.347,55.100,160.011
C01618=1017.166,37.659,-109.890,166.344,55.108,160.012
C01619=1017.161,37.409,-109.876,166.342,55.116,160.013
C01620=1017.155,37.159,-109.861,166.338,55.124,160.013
C01621=1017.150,36.910,-109.846,166.335,55.131,160.014
C01622=1017.145,36.660,-109.831,166.333,55.139,160.015
C01623=1017.140,36.411,-109.816,166.330,55.147,160.016
C01624=1017.134,36.162,-109.802,166.328,55.155,160.017
C01625=1017.129,35.911,-109.787,166.326,55.163,160.018
C01626=1017.123,35.663,-109.772,166.323,55.171,160.019
C01627=1017.118,35.413,-109.758,166.321,55.179,160.020
C01628=1017.113,35.164,-109.743,166.317,55.187,160.021
C01629=1017.108,34.914,-109.729,166.315,55.195,160.022
C01630=1017.102,34.665,-109.714,166.312,55.202,160.023
C01631=1017.097,34.415,-109.700,166.310,55.210,160.024
C01632=1017.091,34.165,-109.685,166.308,55.218,160.025
C01633=1017.086,33.915,-109.670,166.305,55.226,160.026
C01634=1017.081,33.666,-109.656,166.303,55.234,160.027
C01635=1017.076,33.417,-109.641,166.299,55.242,160.027
C01636=1017.070,33.168,-109.627,166.297,55.250,160.028
C01637=1017.065,32.918,-109.613,166.295,55.258,160.029
C01638=1017.059,32.669,-109.598,166.292,55.266,160.030
C01639=1017.054,32.419,-109.584,166.290,55.273,160.031
C01640=1017.049,32.169,-109.569,166.288,55.281,160.032
C01641=1017.043,31.920,-109.554,166.285,55.289,160.033
C01642=1017.038,31.670,-109.540,166.281,55.297,160.034
C01643=1017.032,31.421,-109.525,166.279,55.305,160.035
C01644=1017.028,31.171,-109.511,166.276,55.312,160.036
C01645=1017.022,30.922,-109.496,166.274,55.321,160.037
C01646=1017.017,30.672,-109.482,166.271,55.328,160.037
C01647=1017.012,30.422,-109.468,166.269,55.336,160.039
C01648=1017.007,30.173,-109.453,166.267,55.344,160.039
C01649=1017.001,29.924,-109.439,166.264,55.352,160.040
C01650=1016.996,29.674,-109.424,166.262,55.359,160.041
C01651=1016.991,29.425,-109.410,166.259,55.367,160.042
C01652=1016.986,29.175,-109.395,166.256,55.375,160.043
C01653=1016.980,28.926,-109.381,166.253,55.383,160.044
C01654=1016.975,28.676,-109.366,166.251,55.391,160.045
C01655=1016.969,28.426,-109.351,166.248,55.398,160.046
C01656=1016.964,28.177,-109.337,166.246,55.406,160.047
C01657=1016.959,27.927,-109.323,166.244,55.414,160.048
C01658=1016.954,27.678,-109.308,166.241,55.422,160.048
C01659=1016.948,27.428,-109.294,166.238,55.429,160.049
C01660=1016.943,27.179,-109.280,166.236,55.437,160.050
C01661=1016.938,26.896,-109.264,166.233,55.446,160.051
C01662=1016.931,26.615,-109.248,166.230,55.455,160.052
C01663=1016.925,26.332,-109.232,166.227,55.464,160.053
C01664=1016.919,26.050,-109.216,166.224,55.473,160.055
C01665=1016.913,25.801,-109.201,166.222,55.481,160.055
C01666=1016.909,25.551,-109.187,166.220,55.489,160.056
C01667=1016.903,25.302,-109.173,166.216,55.497,160.057
C01668=1016.898,25.052,-109.159,166.213,55.504,160.058
C01669=1016.893,24.802,-109.145,166.211,55.512,160.059
C01670=1016.887,24.552,-109.131,166.209,55.520,160.060
C01671=1016.882,24.304,-109.116,166.206,55.528,160.061
C01672=1016.876,24.054,-109.102,166.204,55.536,160.062
C01673=1016.871,23.804,-109.089,166.201,55.544,160.063
C01674=1016.866,23.554,-109.074,166.198,55.552,160.063
C01675=1016.860,23.305,-109.060,166.195,55.559,160.064
C01676=1016.855,23.055,-109.046,166.193,55.567,160.065
C01677=1016.849,22.806,-109.033,166.191,55.575,160.066
C01678=1016.845,22.556,-109.018,166.189,55.583,160.067
C01679=1016.839,22.307,-109.004,166.186,55.591,160.068
C01680=1016.833,22.057,-108.990,166.182,55.599,160.069
C01681=1016.828,21.808,-108.976,166.180,55.607,160.070
C01682=1016.824,21.559,-108.962,166.177,55.614,160.071
C01683=1016.818,21.309,-108.948,166.175,55.622,160.072
C01684=1016.813,21.059,-108.934,166.173,55.630,160.073
C01685=1016.807,20.810,-108.920,166.170,55.637,160.073
C01686=1016.802,20.560,-108.906,166.168,55.646,160.075
C01687=1016.797,20.310,-108.892,166.165,55.653,160.075
C01688=1016.792,20.061,-108.878,166.163,55.661,160.076
C01689=1016.786,19.811,-108.864,166.160,55.669,160.077
C01690=1016.781,19.562,-108.850,166.157,55.677,160.078
C01691=1016.776,19.312,-108.836,166.154,55.684,160.079
C01692=1016.771,19.062,-108.822,166.152,55.692,160.080
C01693=1016.765,18.813,-108.808,166.150,55.700,160.081
C01694=1016.760,18.564,-108.794,166.147,55.708,160.081
C01695=1016.755,18.314,-108.781,166.145,55.716,160.083
C01696=1016.749,18.065,-108.767,166.141,55.724,160.083
C01697=1016.744,17.815,-108.753,166.139,55.731,160.084
C01698=1016.738,17.565,-108.739,166.137,55.739,160.085
C01699=1016.733,17.316,-108.725,166.134,55.747,160.086
C01700=1016.727,17.066,-108.711,166.131,55.755,160.087
C01701=1016.722,16.817,-108.697,166.129,55.763,160.088
C01702=1016.718,16.568,-108.683,166.127,55.770,160.089
C01703=1016.713,16.317,-108.670,166.123,55.778,160.089
C01704=1016.707,16.068,-108.656,166.121,55.786,160.090
C01705=1016.702,15.818,-108.642,166.118,55.794,160.091
C01706=1016.696,15.569,-108.629,166.116,55.802,160.092
C01707=1016.691,15.319,-108.615,166.114,55.810,160.093
C01708=1016.686,15.070,-108.601,166.111,55.817,160.094
C01709=1016.680,14.821,-108.587,166.109,55.825,160.095
C01710=1016.675,14.571,-108.574,166.105,55.833,160.096
C01711=1016.670,14.321,-108.560,166.103,55.841,160.097
C01712=1016.664,14.071,-108.547,166.100,55.849,160.097
C01713=1016.659,13.822,-108.533,166.098,55.856,160.098
C01714=1016.654,13.573,-108.519,166.095,55.864,160.099
C01715=1016.649,13.323,-108.506,166.093,55.872,160.100
C01716=1016.643,13.073,-108.492,166.090,55.879,160.101
C01717=1016.638,12.823,-108.478,166.088,55.887,160.102
C01718=1016.632,12.574,-108.464,166.085,55.896,160.103
C01719=1016.627,12.324,-108.451,166.082,55.903,160.104
C01720=1016.622,12.075,-108.438,166.080,55.911,160.105
C01721=1016.616,11.825,-108.425,166.078,55.919,160.106
C01722=1016.611,11.575,-108.411,166.074,55.927,160.106
C01723=1016.605,11.326,-108.397,166.072,55.935,160.107
C01724=1016.600,11.076,-108.384,166.069,55.943,160.108
C01725=1016.594,10.796,-108.369,166.067,55.952,160.109
C01726=1016.588,10.515,-108.355,166.064,55.961,160.110
C01727=1016.582,10.234,-108.339,166.061,55.969,160.111
C01728=1016.576,9.953,-108.325,166.057,55.978,160.112
C01729=1016.571,9.704,-108.311,166.055,55.986,160.113
C01730=1016.565,9.454,-108.297,166.053,55.994,160.114
C01731=1016.560,9.205,-108.285,166.049,56.002,160.115
C01732=1016.554,8.956,-108.271,166.047,56.010,160.116
C01733=1016.549,8.705,-108.258,166.045,56.018,160.117
C01734=1016.544,8.457,-108.244,166.042,56.025,160.117
C01735=1016.538,8.207,-108.232,166.040,56.034,160.119
C01736=1016.533,7.957,-108.218,166.036,56.042,160.119
C01737=1016.528,7.707,-108.205,166.034,56.049,160.120
C01738=1016.523,7.458,-108.191,166.031,56.057,160.121
C01739=1016.518,7.208,-108.178,166.029,56.065,160.122
C01740=1016.511,6.959,-108.165,166.027,56.072,160.123
C01741=1016.507,6.710,-108.151,166.023,56.080,160.123
C01742=1016.501,6.459,-108.138,166.021,56.088,160.124
C01743=1016.496,6.210,-108.124,166.019,56.096,160.125
C01744=1016.490,5.960,-108.112,166.016,56.104,160.126
C01745=1016.485,5.711,-108.098,166.014,56.111,160.127
C01746=1016.480,5.461,-108.085,166.011,56.119,160.128
C01747=1016.475,5.211,-108.072,166.008,56.128,160.129
C01748=1016.469,4.962,-108.059,166.005,56.135,160.130
C01749=1016.464,4.712,-108.046,166.003,56.143,160.130
C01750=1016.459,4.462,-108.032,166.000,56.150,160.131
C01751=1016.454,4.213,-108.019,165.998,56.158,160.132
C01752=1016.448,3.964,-108.006,165.995,56.166,160.133
C01753=1016.443,3.714,-107.993,165.993,56.174,160.134
C01754=1016.438,3.465,-107.979,165.990,56.182,160.135
C01755=1016.433,3.214,-107.966,165.987,56.189,160.136
C01756=1016.427,2.965,-107.954,165.985,56.197,160.136
C01757=1016.422,2.716,-107.940,165.982,56.205,160.137
C01758=1016.417,2.465,-107.927,165.979,56.212,160.138
C01759=1016.412,2.217,-107.913,165.977,56.220,160.139
C01760=1016.407,1.966,-107.900,165.974,56.227,160.140
C01761=1016.401,1.718,-107.887,165.972,56.236,160.141
C01762=1016.396,1.468,-107.874,165.969,56.244,160.141
C01763=1016.391,1.217,-107.861,165.966,56.251,160.142
C01764=1016.386,0.969,-107.848,165.964,56.259,160.143
C01765=1016.380,0.719,-107.835,165.961,56.266,160.144
C01766=1016.375,0.469,-107.822,165.959,56.274,160.145
C01767=1016.370,0.220,-107.808,165.956,56.281,160.146
C01768=1016.365,-0.031,-107.795,165.954,56.289,160.147
C01769=1016.359,-0.280,-107.783,165.951,56.297,160.147
C01770=1016.354,-0.529,-107.769,165.949,56.304,160.148
C01771=1016.349,-0.779,-107.756,165.946,56.312,160.149
C01772=1016.344,-1.029,-107.743,165.943,56.320,160.150
C01773=1016.339,-1.278,-107.730,165.940,56.327,160.150
C01774=1016.333,-1.528,-107.717,165.938,56.335,160.151
C01775=1016.329,-1.777,-107.704,165.935,56.343,160.152
C01776=1016.323,-2.027,-107.691,165.933,56.350,160.153
C01777=1016.317,-2.277,-107.678,165.930,56.358,160.154
C01778=1016.313,-2.526,-107.665,165.928,56.365,160.155
C01779=1016.307,-2.776,-107.651,165.925,56.373,160.156
C01780=1016.303,-3.025,-107.639,165.923,56.381,160.156
C01781=1016.297,-3.275,-107.626,165.920,56.388,160.157
C01782=1016.292,-3.525,-107.613,165.918,56.396,160.158
C01783=1016.287,-3.774,-107.599,165.915,56.403,160.159
C01784=1016.282,-4.023,-107.587,165.912,56.410,160.159
C01785=1016.276,-4.274,-107.574,165.910,56.418,160.160
